C03641=1053.652,-40.489,430.295,170.687,30.205,155.689
C03642=1053.645,-40.738,430.307,170.685,30.204,155.689
C03643=1053.639,-40.988,430.320,170.683,30.202,155.688
C03644=1053.633,-41.237,430.333,170.681,30.201,155.688
C03645=1053.627,-41.487,430.346,170.680,30.199,155.688
C03646=1053.620,-41.736,430.359,170.678,30.197,155.688
C03647=1053.615,-41.986,430.372,170.676,30.195,155.688
C03648=1053.607,-42.236,430.385,170.674,30.194,155.687
C03649=1053.601,-42.485,430.397,170.672,30.192,155.687
C03650=1053.595,-42.735,430.410,170.670,30.191,155.687
C03651=1053.589,-42.985,430.423,170.669,30.189,155.687
C03652=1053.583,-43.234,430.436,170.667,30.188,155.687
C03653=1053.576,-43.483,430.448,170.665,30.185,155.687
C03654=1053.570,-43.733,430.461,170.663,30.184,155.686
C03655=1053.564,-43.983,430.474,170.661,30.182,155.686
C03656=1053.558,-44.233,430.487,170.660,30.181,155.686
C03657=1053.551,-44.482,430.499,170.658,30.179,155.686
C03658=1053.545,-44.731,430.512,170.656,30.178,155.686
C03659=1053.539,-44.981,430.524,170.654,30.176,155.686
C03660=1053.533,-45.230,430.538,170.652,30.174,155.685
C03661=1053.527,-45.480,430.550,170.650,30.172,155.685
C03662=1053.521,-45.730,430.562,170.649,30.171,155.685
C03663=1053.514,-45.979,430.575,170.647,30.169,155.685
C03664=1053.508,-46.229,430.588,170.645,30.168,155.685
C03665=1053.503,-46.479,430.601,170.643,30.166,155.685
C03666=1053.496,-46.728,430.613,170.641,30.164,155.684
C03667=1053.490,-46.978,430.626,170.639,30.163,155.684
C03668=1053.484,-47.228,430.638,170.638,30.161,155.684
C03669=1053.478,-47.478,430.651,170.636,30.160,155.684
C03670=1053.471,-47.727,430.664,170.634,30.158,155.684
C03671=1053.465,-47.976,430.676,170.632,30.157,155.684
C03672=1053.459,-48.226,430.689,170.630,30.154,155.683
C03673=1053.453,-48.476,430.702,170.628,30.153,155.683
C03674=1053.446,-48.725,430.714,170.627,30.151,155.683
C03675=1053.440,-48.975,430.726,170.625,30.150,155.683
C03676=1053.434,-49.225,430.739,170.623,30.148,155.683
C03677=1053.429,-49.474,430.751,170.621,30.147,155.683
C03678=1053.422,-49.723,430.764,170.619,30.145,155.682
C03679=1053.416,-49.973,430.776,170.617,30.143,155.682
C03680=1053.410,-50.223,430.789,170.616,30.142,155.682
C03681=1053.404,-50.504,430.803,170.613,30.140,155.682
C03682=1053.396,-50.783,430.817,170.611,30.139,155.682
C03683=1053.388,-51.064,430.831,170.609,30.137,155.682
C03684=1053.381,-51.344,430.845,170.607,30.135,155.681
C03685=1053.375,-51.594,430.857,170.605,30.134,155.681
C03686=1053.369,-51.844,430.869,170.604,30.132,155.681
C03687=1053.363,-52.093,430.881,170.601,30.130,155.681
C03688=1053.357,-52.343,430.893,170.599,30.129,155.681
C03689=1053.350,-52.592,430.905,170.597,30.127,155.681
C03690=1053.343,-52.841,430.918,170.595,30.126,155.681
C03691=1053.337,-53.091,430.931,170.593,30.125,155.680
C03692=1053.331,-53.341,430.943,170.592,30.123,155.680
C03693=1053.325,-53.590,430.955,170.590,30.122,155.680
C03694=1053.318,-53.840,430.967,170.588,30.120,155.680
C03695=1053.312,-54.090,430.980,170.586,30.119,155.680
C03696=1053.306,-54.339,430.992,170.584,30.118,155.680
C03697=1053.299,-54.589,431.003,170.582,30.116,155.680
C03698=1053.293,-54.839,431.016,170.581,30.114,155.679
C03699=1053.287,-55.088,431.028,170.579,30.113,155.679
C03700=1053.281,-55.338,431.041,170.577,30.112,155.679
C03701=1053.275,-55.587,431.052,170.575,30.110,155.679
C03702=1053.268,-55.837,431.064,170.573,30.109,155.679
C03703=1053.262,-56.087,431.077,170.571,30.107,155.679
C03704=1053.255,-56.336,431.089,170.570,30.106,155.679
C03705=1053.249,-56.586,431.101,170.568,30.105,155.679
C03706=1053.243,-56.836,431.113,170.566,30.103,155.678
C03707=1053.236,-57.085,431.125,170.564,30.101,155.678
C03708=1053.230,-57.335,431.138,170.561,30.100,155.678
C03709=1053.224,-57.584,431.149,170.559,30.099,155.678
C03710=1053.218,-57.834,431.161,170.557,30.097,155.678
C03711=1053.212,-58.084,431.174,170.556,30.096,155.678
C03712=1053.205,-58.334,431.185,170.554,30.094,155.678
C03713=1053.199,-58.583,431.197,170.552,30.093,155.678
C03714=1053.193,-58.833,431.210,170.550,30.091,155.677
C03715=1053.187,-59.082,431.221,170.548,30.090,155.677
C03716=1053.181,-59.332,431.234,170.546,30.088,155.677
C03717=1053.174,-59.581,431.246,170.545,30.087,155.677
C03718=1053.168,-59.831,431.258,170.543,30.086,155.677
C03719=1053.162,-60.081,431.270,170.541,30.084,155.677
C03720=1053.155,-60.331,431.281,170.539,30.083,155.677
C03721=1053.149,-60.580,431.293,170.537,30.082,155.677
C03722=1053.143,-60.830,431.306,170.535,30.080,155.676
C03723=1053.137,-61.079,431.317,170.534,30.079,155.676
C03724=1053.130,-61.329,431.329,170.532,30.078,155.676
C03725=1053.125,-61.578,431.342,170.530,30.076,155.676
C03726=1053.118,-61.828,431.353,170.527,30.074,155.676
C03727=1053.112,-62.078,431.365,170.525,30.073,155.676
C03728=1053.106,-62.328,431.377,170.523,30.072,155.676
C03729=1053.100,-62.577,431.389,170.521,30.070,155.676
C03730=1053.093,-62.827,431.400,170.520,30.069,155.675
C03731=1053.088,-63.077,431.413,170.518,30.068,155.675
C03732=1053.081,-63.326,431.425,170.516,30.066,155.675
C03733=1053.075,-63.575,431.436,170.514,30.064,155.675
C03734=1053.069,-63.826,431.448,170.512,30.063,155.675
C03735=1053.063,-64.075,431.460,170.510,30.062,155.675
C03736=1053.056,-64.325,431.472,170.509,30.060,155.675
C03737=1053.050,-64.574,431.484,170.507,30.059,155.675
C03738=1053.044,-64.824,431.496,170.505,30.058,155.675
C03739=1053.038,-65.074,431.507,170.503,30.056,155.674
C03740=1053.032,-65.323,431.519,170.500,30.055,155.674
C03741=1053.026,-65.573,431.531,170.498,30.053,155.674
C03742=1053.019,-65.823,431.543,170.496,30.052,155.674
C03743=1053.013,-66.072,431.554,170.495,30.051,155.674
C03744=1053.008,-66.322,431.566,170.493,30.049,155.674
C03745=1053.001,-66.570,431.578,170.491,30.048,155.674
C03746=1052.995,-66.819,431.590,170.489,30.047,155.674
C03747=1052.989,-67.068,431.601,170.487,30.045,155.674
C03748=1052.982,-67.317,431.613,170.485,30.044,155.673
C03749=1052.976,-67.565,431.625,170.484,30.043,155.673
C03750=1052.971,-67.813,431.636,170.482,30.042,155.673
C03751=1052.965,-68.062,431.648,170.480,30.040,155.673
C03752=1052.959,-68.311,431.660,170.478,30.038,155.673
C03753=1052.952,-68.560,431.671,170.476,30.038,155.673
C03754=1052.947,-68.810,431.683,170.474,30.036,155.673
C03755=1052.940,-69.060,431.695,170.471,30.035,155.673
C03756=1052.934,-69.310,431.706,170.470,30.033,155.673
C03757=1052.928,-69.559,431.718,170.468,30.032,155.672
C03758=1052.922,-69.809,431.730,170.466,30.031,155.672
C03759=1052.916,-70.058,431.741,170.464,30.029,155.672
C03760=1052.910,-70.308,431.753,170.462,30.028,155.672
C03761=1052.903,-70.558,431.764,170.460,30.027,155.672
C03762=1052.898,-70.807,431.777,170.459,30.026,155.672
C03763=1052.892,-71.057,431.788,170.457,30.024,155.672
C03764=1052.886,-71.306,431.799,170.455,30.023,155.672
C03765=1052.879,-71.556,431.811,170.453,30.021,155.672
C03766=1052.874,-71.806,431.823,170.451,30.020,155.671
C03767=1052.868,-72.056,431.834,170.448,30.019,155.671
C03768=1052.861,-72.305,431.846,170.447,30.017,155.671
C03769=1052.855,-72.555,431.857,170.445,30.016,155.671
C03770=1052.849,-72.805,431.868,170.443,30.015,155.671
C03771=1052.844,-73.054,431.880,170.441,30.014,155.671
C03772=1052.837,-73.304,431.892,170.439,30.012,155.671
C03773=1052.831,-73.553,431.903,170.437,30.011,155.671
C03774=1052.825,-73.803,431.914,170.435,30.009,155.671
C03775=1052.819,-74.052,431.926,170.434,30.008,155.671
C03776=1052.812,-74.302,431.937,170.432,30.007,155.671
C03777=1052.807,-74.552,431.948,170.430,30.006,155.671
C03778=1052.800,-74.802,431.960,170.427,30.005,155.670
C03779=1052.794,-75.052,431.971,170.425,30.003,155.670
C03780=1052.788,-75.301,431.982,170.423,30.002,155.670
C03781=1052.781,-75.551,431.994,170.421,30.001,155.670
C03782=1052.776,-75.800,432.005,170.420,30.000,155.670
C03783=1052.769,-76.050,432.016,170.418,29.999,155.670
C03784=1052.763,-76.299,432.028,170.416,29.998,155.670
C03785=1052.757,-76.550,432.039,170.414,29.996,155.670
C03786=1052.751,-76.799,432.050,170.412,29.995,155.670
C03787=1052.744,-77.049,432.062,170.409,29.994,155.670
C03788=1052.739,-77.298,432.073,170.407,29.992,155.670
C03789=1052.732,-77.582,432.085,170.406,29.991,155.670
C03790=1052.725,-77.866,432.098,170.403,29.990,155.670
C03791=1052.717,-78.149,432.112,170.401,29.989,155.669
C03792=1052.710,-78.433,432.124,170.399,29.988,155.669
C03793=1052.705,-78.683,432.135,170.397,29.986,155.669
C03794=1052.698,-78.933,432.146,170.394,29.985,155.669
C03795=1052.692,-79.182,432.158,170.392,29.984,155.669
C03796=1052.686,-79.432,432.169,170.391,29.982,155.669
C03797=1052.680,-79.682,432.180,170.389,29.981,155.669
C03798=1052.674,-79.931,432.191,170.387,29.981,155.669
C03799=1052.668,-80.181,432.202,170.385,29.980,155.669
C03800=1052.661,-80.430,432.213,170.383,29.979,155.669
C03801=1052.655,-80.680,432.224,170.381,29.978,155.669
C03802=1052.649,-80.930,432.236,170.378,29.976,155.669
C03803=1052.642,-81.180,432.246,170.377,29.975,155.669
C03804=1052.636,-81.430,432.257,170.375,29.974,155.669
C03805=1052.630,-81.679,432.268,170.373,29.973,155.669
C03806=1052.624,-81.929,432.279,170.371,29.972,155.669
C03807=1052.617,-82.179,432.290,170.369,29.971,155.669
C03808=1052.611,-82.427,432.301,170.367,29.970,155.668
C03809=1052.604,-82.711,432.314,170.364,29.969,155.668
C03810=1052.597,-82.995,432.326,170.363,29.967,155.668
C03811=1052.589,-83.279,432.338,170.360,29.966,155.668
C03812=1052.582,-83.563,432.351,170.358,29.965,155.668
C03813=1052.576,-83.813,432.362,170.356,29.964,155.668
C03814=1052.569,-84.063,432.373,170.354,29.963,155.668
C03815=1052.564,-84.312,432.384,170.352,29.962,155.668
C03816=1052.558,-84.562,432.394,170.349,29.961,155.668
C03817=1052.552,-84.812,432.406,170.347,29.960,155.668
C03818=1052.545,-85.061,432.416,170.346,29.959,155.668
C03819=1052.539,-85.311,432.427,170.344,29.958,155.668
C03820=1052.533,-85.561,432.438,170.342,29.957,155.668
C03821=1052.527,-85.810,432.448,170.340,29.956,155.668
C03822=1052.520,-86.060,432.460,170.338,29.955,155.668
C03823=1052.514,-86.309,432.470,170.335,29.954,155.668
C03824=1052.507,-86.559,432.481,170.333,29.953,155.668
C03825=1052.502,-86.809,432.492,170.331,29.952,155.668
C03826=1052.496,-87.058,432.503,170.330,29.951,155.668
C03827=1052.489,-87.308,432.514,170.328,29.950,155.668
C03828=1052.483,-87.558,432.524,170.326,29.949,155.668
C03829=1052.477,-87.808,432.535,170.324,29.948,155.668
C03830=1052.471,-88.058,432.545,170.321,29.947,155.668
C03831=1052.465,-88.307,432.556,170.319,29.946,155.668
C03832=1052.459,-88.557,432.567,170.317,29.945,155.668
C03833=1052.452,-88.807,432.578,170.315,29.944,155.668
C03834=1052.446,-89.056,432.588,170.314,29.943,155.667
C03835=1052.440,-89.306,432.600,170.312,29.942,155.667
C03836=1052.433,-89.555,432.610,170.309,29.941,155.667
C03837=1052.428,-89.805,432.621,170.307,29.940,155.667
C03838=1052.422,-90.056,432.631,170.305,29.939,155.667
C03839=1052.415,-90.305,432.642,170.303,29.938,155.667
C03840=1052.409,-90.554,432.653,170.301,29.937,155.667
C03841=1052.404,-90.804,432.663,170.300,29.936,155.667
C03842=1052.397,-91.054,432.674,170.298,29.935,155.667
C03843=1052.391,-91.303,432.685,170.295,29.934,155.667
C03844=1052.385,-91.553,432.695,170.293,29.933,155.667
C03845=1052.378,-91.803,432.706,170.291,29.932,155.667
C03846=1052.373,-92.053,432.717,170.289,29.932,155.667
C03847=1052.366,-92.302,432.727,170.287,29.931,155.667
C03848=1052.360,-92.551,432.738,170.285,29.930,155.667
C03849=1052.354,-92.802,432.748,170.283,29.929,155.667
C03850=1052.348,-93.051,432.759,170.281,29.928,155.667
C03851=1052.342,-93.301,432.770,170.279,29.927,155.667
C03852=1052.336,-93.550,432.780,170.277,29.926,155.667
C03853=1052.330,-93.801,432.790,170.275,29.925,155.667
C03854=1052.324,-94.050,432.801,170.273,29.924,155.667
C03855=1052.317,-94.299,432.811,170.271,29.923,155.667
C03856=1052.312,-94.550,432.822,170.268,29.922,155.667
C03857=1052.305,-94.799,432.832,170.267,29.921,155.667
C03858=1052.299,-95.049,432.843,170.265,29.920,155.667
C03859=1052.293,-95.298,432.854,170.263,29.919,155.667
C03860=1052.287,-95.548,432.864,170.261,29.918,155.667
C03861=1052.282,-95.798,432.874,170.259,29.918,155.667
C03862=1052.274,-96.048,432.885,170.257,29.917,155.667
C03863=1052.269,-96.298,432.895,170.254,29.916,155.667
C03864=1052.263,-96.547,432.906,170.252,29.915,155.667
C03865=1052.257,-96.796,432.916,170.250,29.914,155.667
C03866=1052.251,-97.047,432.927,170.249,29.913,155.667
C03867=1052.244,-97.296,432.937,170.247,29.912,155.667
C03868=1052.239,-97.547,432.947,170.245,29.911,155.667
C03869=1052.232,-97.796,432.958,170.242,29.910,155.667
C03870=1052.227,-98.045,432.969,170.240,29.910,155.667
C03871=1052.221,-98.295,432.978,170.238,29.909,155.667
C03872=1052.213,-98.545,432.989,170.236,29.908,155.667
C03873=1052.206,-98.831,433.000,170.233,29.907,155.667
C03874=1052.199,-99.117,433.012,170.232,29.906,155.667
C03875=1052.193,-99.403,433.024,170.229,29.905,155.667
C03876=1052.186,-99.689,433.036,170.227,29.904,155.667
C03877=1052.180,-99.939,433.045,170.225,29.904,155.667
C03878=1052.173,-100.189,433.056,170.223,29.903,155.667
C03879=1052.167,-100.438,433.067,170.220,29.902,155.667
C03880=1052.161,-100.688,433.076,170.218,29.901,155.667
C03881=1052.154,-100.937,433.087,170.216,29.901,155.667
C03882=1052.149,-101.187,433.097,170.214,29.900,155.667
C03883=1052.143,-101.437,433.106,170.213,29.899,155.667
C03884=1052.136,-101.687,433.117,170.211,29.899,155.667
C03885=1052.130,-101.937,433.127,170.208,29.898,155.667
C03886=1052.124,-102.186,433.138,170.206,29.897,155.667
C03887=1052.118,-102.436,433.147,170.204,29.896,155.667
C03888=1052.112,-102.686,433.158,170.202,29.895,155.667
C03889=1052.106,-102.935,433.168,170.200,29.895,155.667
C03890=1052.099,-103.185,433.178,170.197,29.894,155.667
C03891=1052.094,-103.435,433.188,170.195,29.893,155.667
C03892=1052.087,-103.685,433.198,170.194,29.892,155.667
C03893=1052.081,-103.934,433.208,170.192,29.892,155.667
C03894=1052.074,-104.184,433.218,170.190,29.891,155.667
C03895=1052.069,-104.434,433.229,170.188,29.891,155.667
C03896=1052.063,-104.683,433.238,170.185,29.890,155.667
C03897=1052.056,-104.933,433.248,170.183,29.889,155.667
C03898=1052.051,-105.183,433.259,170.181,29.888,155.667
C03899=1052.044,-105.433,433.268,170.179,29.888,155.667
C03900=1052.038,-105.682,433.278,170.177,29.887,155.667
C03901=1052.032,-105.931,433.288,170.174,29.886,155.667
C03902=1052.026,-106.182,433.298,170.173,29.885,155.667
C03903=1052.020,-106.431,433.308,170.171,29.885,155.667
C03904=1052.014,-106.681,433.318,170.169,29.884,155.667
C03905=1052.007,-106.931,433.328,170.167,29.884,155.667
C03906=1052.002,-107.181,433.338,170.165,29.883,155.667
C03907=1051.995,-107.431,433.348,170.162,29.882,155.667
C03908=1051.989,-107.680,433.358,170.160,29.882,155.668
C03909=1051.983,-107.930,433.368,170.158,29.881,155.667
C03910=1051.977,-108.180,433.377,170.156,29.880,155.668
C03911=1051.970,-108.430,433.387,170.154,29.879,155.668
C03912=1051.964,-108.679,433.397,170.152,29.879,155.668
C03913=1051.958,-108.929,433.407,170.150,29.879,155.668
C03914=1051.952,-109.179,433.417,170.148,29.878,155.668
C03915=1051.946,-109.428,433.426,170.146,29.877,155.668
C03916=1051.940,-109.678,433.436,170.144,29.877,155.668
C03917=1051.933,-109.927,433.446,170.141,29.876,155.668
C03918=1051.927,-110.177,433.456,170.139,29.875,155.668
C03919=1051.921,-110.427,433.465,170.137,29.875,155.668
C03920=1051.915,-110.677,433.475,170.135,29.875,155.668
C03921=1051.909,-110.927,433.484,170.133,29.874,155.668
C03922=1051.903,-111.176,433.495,170.131,29.873,155.668
C03923=1051.897,-111.426,433.505,170.129,29.873,155.668
C03924=1051.891,-111.676,433.514,170.127,29.872,155.668
C03925=1051.885,-111.926,433.524,170.125,29.871,155.668
C03926=1051.878,-112.175,433.534,170.123,29.871,155.668
C03927=1051.872,-112.425,433.543,170.120,29.870,155.668
C03928=1051.866,-112.675,433.553,170.118,29.869,155.668
C03929=1051.860,-112.925,433.562,170.116,29.869,155.668
C03930=1051.854,-113.174,433.572,170.114,29.869,155.668
C03931=1051.847,-113.424,433.582,170.112,29.868,155.669
C03932=1051.841,-113.673,433.592,170.109,29.867,155.669
C03933=1051.835,-113.923,433.601,170.108,29.867,155.669
C03934=1051.829,-114.173,433.611,170.106,29.866,155.669
C03935=1051.823,-114.423,433.621,170.104,29.866,155.669
C03936=1051.817,-114.673,433.631,170.102,29.866,155.669
C03937=1051.810,-114.957,433.641,170.099,29.865,155.669
C03938=1051.803,-115.242,433.651,170.097,29.864,155.669
C03939=1051.796,-115.526,433.663,170.094,29.864,155.669
C03940=1051.789,-115.811,433.673,170.092,29.863,155.669
C03941=1051.783,-116.061,433.683,170.089,29.863,155.669
C03942=1051.776,-116.311,433.693,170.087,29.862,155.669
C03943=1051.770,-116.561,433.702,170.085,29.862,155.669
C03944=1051.764,-116.811,433.712,170.083,29.862,155.669
C03945=1051.758,-117.060,433.721,170.082,29.861,155.669
C03946=1051.752,-117.310,433.730,170.079,29.860,155.670
C03947=1051.746,-117.559,433.740,170.077,29.860,155.670
C03948=1051.740,-117.809,433.750,170.075,29.859,155.670
C03949=1051.734,-118.060,433.758,170.073,29.859,155.670
C03950=1051.728,-118.309,433.768,170.071,29.859,155.670
C03951=1051.722,-118.559,433.778,170.068,29.858,155.670
C03952=1051.716,-118.809,433.787,170.066,29.858,155.670
C03953=1051.709,-119.058,433.796,170.064,29.857,155.670
C03954=1051.702,-119.308,433.806,170.062,29.857,155.670
C03955=1051.697,-119.557,433.815,170.060,29.857,155.670
C03956=1051.691,-119.807,433.824,170.057,29.856,155.670
C03957=1051.685,-120.057,433.834,170.056,29.856,155.670
C03958=1051.679,-120.307,433.843,170.054,29.855,155.670
C03959=1051.673,-120.557,433.852,170.052,29.855,155.671
C03960=1051.666,-120.807,433.862,170.049,29.855,155.671
C03961=1051.660,-121.057,433.872,170.047,29.854,155.671
C03962=1051.654,-121.306,433.880,170.045,29.854,155.671
C03963=1051.648,-121.555,433.890,170.043,29.853,155.671
C03964=1051.642,-121.806,433.899,170.041,29.853,155.671
C03965=1051.636,-122.056,433.908,170.038,29.853,155.671
C03966=1051.629,-122.305,433.918,170.036,29.852,155.671
C03967=1051.624,-122.554,433.927,170.034,29.852,155.671
C03968=1051.617,-122.804,433.936,170.032,29.851,155.671
C03969=1051.611,-123.054,433.945,170.030,29.851,155.671
C03970=1051.605,-123.304,433.954,170.028,29.851,155.671
C03971=1051.599,-123.554,433.964,170.026,29.850,155.672
C03972=1051.593,-123.803,433.973,170.024,29.850,155.672
C03973=1051.587,-124.053,433.982,170.022,29.850,155.672
C03974=1051.580,-124.303,433.991,170.020,29.850,155.672
C03975=1051.574,-124.553,434.000,170.017,29.849,155.672
C03976=1051.568,-124.803,434.009,170.015,29.849,155.672
C03977=1051.563,-125.052,434.018,170.013,29.848,155.672
C03978=1051.556,-125.302,434.027,170.011,29.848,155.672
C03979=1051.550,-125.552,434.036,170.008,29.848,155.672
C03980=1051.544,-125.802,434.046,170.006,29.848,155.672
C03981=1051.537,-126.051,434.055,170.004,29.847,155.673
C03982=1051.532,-126.301,434.063,170.002,29.847,155.673
C03983=1051.526,-126.551,434.073,170.000,29.847,155.673
C03984=1051.519,-126.801,434.082,169.998,29.847,155.673
C03985=1051.513,-127.051,434.091,169.996,29.846,155.673
C03986=1051.507,-127.300,434.100,169.994,29.846,155.673
C03987=1051.501,-127.550,434.109,169.992,29.846,155.673
C03988=1051.494,-127.800,434.118,169.989,29.845,155.673
C03989=1051.490,-128.049,434.128,169.987,29.845,155.673
C03990=1051.486,-128.299,434.138,169.985,29.844,155.673
C03991=1051.482,-128.550,434.148,169.983,29.842,155.673
C03992=1051.480,-128.799,434.159,169.981,29.840,155.673
C03993=1051.479,-129.050,434.172,169.981,29.837,155.672
C03994=1051.480,-129.301,434.185,169.979,29.834,155.672
C03995=1051.481,-129.551,434.198,169.977,29.830,155.672
C03996=1051.483,-129.801,434.213,169.977,29.826,155.671
C03997=1051.486,-130.052,434.227,169.975,29.822,155.670
C03998=1051.491,-130.302,434.243,169.975,29.817,155.669
C03999=1051.497,-130.553,434.259,169.974,29.811,155.668
C04000=1051.503,-130.803,434.275,169.974,29.805,155.667
C04001=1051.137,-130.826,434.054,169.927,29.973,155.700
C04002=1051.131,-130.577,434.037,169.928,29.980,155.701
C04003=1051.125,-130.326,434.021,169.928,29.985,155.702
C04004=1051.120,-130.076,434.006,169.929,29.990,155.703
C04005=1051.117,-129.824,433.990,169.930,29.995,155.703
C04006=1051.114,-129.574,433.977,169.931,29.999,155.704
C04007=1051.113,-129.324,433.962,169.933,30.003,155.704
C04008=1051.113,-129.074,433.951,169.934,30.006,155.705
C04009=1051.114,-128.823,433.938,169.935,30.008,155.705
C04010=1051.116,-128.573,433.927,169.937,30.010,155.705
C04011=1051.119,-128.323,433.916,169.939,30.012,155.706
C04012=1051.123,-128.073,433.905,169.941,30.013,155.706
C04013=1051.128,-127.823,433.897,169.943,30.014,155.706
C04014=1051.134,-127.573,433.887,169.945,30.015,155.706
C04015=1051.140,-127.324,433.878,169.947,30.014,155.705
C04016=1051.146,-127.074,433.870,169.949,30.015,155.705
C04017=1051.153,-126.824,433.860,169.951,30.015,155.705
C04018=1051.159,-126.575,433.851,169.954,30.016,155.705
C04019=1051.165,-126.324,433.842,169.956,30.015,155.705
C04020=1051.171,-126.075,433.833,169.958,30.016,155.705
C04021=1051.177,-125.826,433.823,169.960,30.016,155.705
C04022=1051.183,-125.575,433.815,169.962,30.016,155.705
C04023=1051.190,-125.326,433.806,169.965,30.017,155.705
C04024=1051.196,-125.076,433.796,169.967,30.017,155.704
C04025=1051.201,-124.826,433.788,169.969,30.017,155.704
C04026=1051.207,-124.576,433.778,169.971,30.017,155.704
C04027=1051.214,-124.327,433.769,169.974,30.018,155.704
C04028=1051.220,-124.076,433.760,169.976,30.018,155.704
C04029=1051.226,-123.827,433.751,169.977,30.019,155.704
C04030=1051.232,-123.577,433.741,169.979,30.019,155.704
C04031=1051.238,-123.328,433.732,169.981,30.019,155.704
C04032=1051.245,-123.078,433.724,169.984,30.019,155.704
C04033=1051.251,-122.828,433.714,169.986,30.020,155.704
C04034=1051.257,-122.579,433.705,169.988,30.020,155.704
C04035=1051.263,-122.329,433.695,169.990,30.020,155.703
C04036=1051.269,-122.078,433.686,169.993,30.021,155.703
C04037=1051.275,-121.829,433.677,169.995,30.021,155.703
C04038=1051.282,-121.579,433.668,169.997,30.021,155.703
C04039=1051.288,-121.329,433.658,169.999,30.022,155.703
C04040=1051.293,-121.080,433.649,170.001,30.022,155.703
C04041=1051.300,-120.831,433.640,170.004,30.023,155.703
C04042=1051.305,-120.580,433.631,170.006,30.023,155.703
C04043=1051.312,-120.330,433.621,170.007,30.023,155.703
C04044=1051.318,-120.080,433.612,170.009,30.024,155.703
C04045=1051.324,-119.831,433.602,170.012,30.024,155.703
C04046=1051.330,-119.582,433.593,170.014,30.025,155.703
C04047=1051.336,-119.332,433.584,170.016,30.025,155.703
C04048=1051.343,-119.082,433.574,170.018,30.025,155.702
C04049=1051.348,-118.832,433.565,170.020,30.026,155.702
C04050=1051.355,-118.582,433.556,170.023,30.026,155.702
C04051=1051.361,-118.332,433.546,170.025,30.027,155.702
C04052=1051.367,-118.082,433.537,170.027,30.027,155.702
C04053=1051.373,-117.833,433.527,170.029,30.027,155.702
C04054=1051.379,-117.583,433.518,170.031,30.028,155.702
C04055=1051.385,-117.334,433.508,170.034,30.028,155.702
C04056=1051.391,-117.084,433.499,170.035,30.029,155.702
C04057=1051.397,-116.834,433.489,170.037,30.030,155.702
C04058=1051.403,-116.584,433.480,170.039,30.030,155.702
C04059=1051.410,-116.335,433.471,170.042,30.030,155.702
C04060=1051.416,-116.085,433.461,170.044,30.031,155.702
C04061=1051.423,-115.835,433.452,170.046,30.031,155.701
C04062=1051.429,-115.550,433.440,170.048,30.031,155.701
C04063=1051.436,-115.265,433.430,170.051,30.032,155.701
C04064=1051.443,-114.980,433.419,170.054,30.033,155.701
C04065=1051.451,-114.696,433.408,170.056,30.034,155.701
C04066=1051.457,-114.446,433.398,170.058,30.034,155.701
C04067=1051.463,-114.197,433.389,170.059,30.034,155.701
C04068=1051.469,-113.947,433.379,170.062,30.035,155.701
C04069=1051.475,-113.697,433.370,170.064,30.035,155.701
C04070=1051.481,-113.448,433.360,170.066,30.036,155.701
C04071=1051.487,-113.197,433.350,170.068,30.036,155.701
C04072=1051.493,-112.948,433.341,170.070,30.037,155.701
C04073=1051.499,-112.698,433.331,170.073,30.037,155.701
C04074=1051.505,-112.448,433.321,170.075,30.038,155.701
C04075=1051.511,-112.198,433.312,170.077,30.039,155.701
C04076=1051.517,-111.948,433.302,170.079,30.039,155.701
C04077=1051.524,-111.699,433.292,170.081,30.039,155.701
C04078=1051.530,-111.449,433.282,170.083,30.041,155.701
C04079=1051.536,-111.200,433.273,170.085,30.041,155.700
C04080=1051.542,-110.950,433.263,170.087,30.041,155.700
C04081=1051.549,-110.700,433.254,170.089,30.042,155.700
C04082=1051.554,-110.450,433.244,170.091,30.043,155.700
C04083=1051.560,-110.200,433.234,170.094,30.043,155.700
C04084=1051.567,-109.951,433.224,170.096,30.043,155.700
C04085=1051.573,-109.701,433.214,170.098,30.044,155.700
C04086=1051.579,-109.451,433.205,170.100,30.045,155.700
C04087=1051.585,-109.202,433.195,170.102,30.045,155.700
C04088=1051.591,-108.952,433.185,170.105,30.046,155.700
C04089=1051.598,-108.703,433.175,170.107,30.047,155.700
C04090=1051.604,-108.453,433.166,170.108,30.047,155.700
C04091=1051.609,-108.203,433.155,170.110,30.048,155.700
C04092=1051.616,-107.953,433.146,170.112,30.048,155.700
C04093=1051.622,-107.704,433.136,170.115,30.049,155.700
C04094=1051.628,-107.454,433.126,170.117,30.050,155.700
C04095=1051.634,-107.204,433.116,170.119,30.050,155.700
C04096=1051.641,-106.954,433.107,170.121,30.051,155.700
C04097=1051.647,-106.704,433.096,170.123,30.051,155.700
C04098=1051.653,-106.454,433.086,170.126,30.052,155.700
C04099=1051.659,-106.205,433.077,170.128,30.053,155.700
C04100=1051.666,-105.955,433.066,170.129,30.053,155.700
C04101=1051.671,-105.705,433.056,170.131,30.054,155.700
C04102=1051.677,-105.455,433.047,170.133,30.055,155.700
C04103=1051.684,-105.206,433.036,170.136,30.056,155.700
C04104=1051.690,-104.956,433.027,170.138,30.056,155.700
C04105=1051.695,-104.706,433.017,170.140,30.057,155.700
C04106=1051.702,-104.457,433.006,170.142,30.057,155.699
C04107=1051.708,-104.207,432.997,170.144,30.058,155.700
C04108=1051.714,-103.958,432.986,170.147,30.059,155.699
C04109=1051.721,-103.707,432.976,170.149,30.060,155.699
C04110=1051.727,-103.458,432.966,170.150,30.060,155.699
C04111=1051.732,-103.208,432.955,170.152,30.061,155.699
C04112=1051.739,-102.958,432.946,170.154,30.062,155.699
C04113=1051.745,-102.709,432.936,170.156,30.063,155.699
C04114=1051.751,-102.459,432.926,170.159,30.063,155.699
C04115=1051.757,-102.209,432.916,170.161,30.064,155.699
C04116=1051.763,-101.960,432.906,170.163,30.064,155.699
C04117=1051.769,-101.710,432.896,170.165,30.065,155.699
C04118=1051.776,-101.460,432.885,170.167,30.066,155.699
C04119=1051.782,-101.210,432.875,170.170,30.067,155.699
C04120=1051.788,-100.961,432.865,170.171,30.068,155.699
C04121=1051.794,-100.711,432.855,170.173,30.068,155.699
C04122=1051.800,-100.462,432.844,170.175,30.069,155.699
C04123=1051.806,-100.212,432.835,170.177,30.070,155.699
C04124=1051.813,-99.962,432.824,170.179,30.071,155.699
C04125=1051.819,-99.712,432.814,170.182,30.072,155.699
C04126=1051.826,-99.426,432.802,170.184,30.072,155.699
C04127=1051.833,-99.140,432.791,170.187,30.073,155.699
C04128=1051.840,-98.854,432.779,170.189,30.074,155.699
C04129=1051.848,-98.567,432.767,170.191,30.075,155.699
C04130=1051.853,-98.318,432.756,170.193,30.076,155.699
C04131=1051.860,-98.069,432.746,170.195,30.077,155.699
C04132=1051.865,-97.819,432.736,170.197,30.078,155.699
C04133=1051.872,-97.569,432.726,170.199,30.078,155.699
C04134=1051.879,-97.319,432.716,170.202,30.079,155.699
C04135=1051.884,-97.069,432.705,170.204,30.080,155.699
C04136=1051.890,-96.820,432.694,170.206,30.080,155.699
C04137=1051.896,-96.570,432.685,170.208,30.081,155.699
C04138=1051.902,-96.321,432.674,170.209,30.082,155.699
C04139=1051.909,-96.071,432.663,170.211,30.083,155.699
C04140=1051.914,-95.821,432.653,170.213,30.084,155.699
C04141=1051.920,-95.571,432.642,170.216,30.085,155.699
C04142=1051.927,-95.322,432.632,170.218,30.086,155.699
C04143=1051.932,-95.072,432.622,170.220,30.087,155.699
C04144=1051.939,-94.822,432.611,170.222,30.088,155.699
C04145=1051.945,-94.573,432.600,170.224,30.089,155.699
C04146=1051.951,-94.323,432.590,170.225,30.090,155.699
C04147=1051.957,-94.073,432.580,170.228,30.091,155.699
C04148=1051.963,-93.824,432.569,170.230,30.091,155.699
C04149=1051.970,-93.574,432.558,170.232,30.092,155.699
C04150=1051.975,-93.324,432.548,170.234,30.093,155.699
C04151=1051.981,-93.074,432.537,170.236,30.094,155.699
C04152=1051.987,-92.825,432.527,170.238,30.095,155.699
C04153=1051.994,-92.575,432.515,170.241,30.096,155.699
C04154=1052.000,-92.325,432.506,170.243,30.097,155.700
C04155=1052.006,-92.076,432.495,170.244,30.098,155.700
C04156=1052.012,-91.825,432.484,170.246,30.099,155.700
C04157=1052.018,-91.576,432.473,170.248,30.099,155.700
C04158=1052.024,-91.327,432.463,170.250,30.100,155.700
C04159=1052.030,-91.077,432.452,170.252,30.101,155.700
C04160=1052.037,-90.827,432.442,170.255,30.103,155.700
C04161=1052.042,-90.577,432.431,170.257,30.103,155.700
C04162=1052.049,-90.328,432.421,170.259,30.104,155.700
C04163=1052.055,-90.078,432.409,170.260,30.105,155.700
C04164=1052.061,-89.828,432.399,170.262,30.106,155.700
C04165=1052.067,-89.579,432.389,170.264,30.107,155.700
C04166=1052.073,-89.328,432.378,170.267,30.108,155.700
C04167=1052.079,-89.079,432.367,170.269,30.109,155.700
C04168=1052.086,-88.830,432.357,170.271,30.110,155.700
C04169=1052.092,-88.580,432.345,170.273,30.111,155.700
C04170=1052.098,-88.330,432.334,170.275,30.112,155.700
C04171=1052.104,-88.081,432.324,170.276,30.113,155.700
C04172=1052.111,-87.831,432.313,170.278,30.114,155.700
C04173=1052.116,-87.581,432.302,170.281,30.115,155.700
C04174=1052.123,-87.332,432.292,170.283,30.116,155.700
C04175=1052.129,-87.082,432.280,170.285,30.117,155.700
C04176=1052.135,-86.832,432.270,170.287,30.118,155.700
C04177=1052.142,-86.582,432.260,170.289,30.119,155.700
C04178=1052.147,-86.332,432.249,170.291,30.120,155.700
C04179=1052.153,-86.083,432.238,170.293,30.121,155.700
C04180=1052.160,-85.833,432.227,170.295,30.122,155.700
C04181=1052.166,-85.584,432.216,170.297,30.123,155.700
C04182=1052.172,-85.333,432.205,170.299,30.124,155.700
C04183=1052.179,-85.084,432.195,170.301,30.125,155.700
C04184=1052.184,-84.835,432.184,170.303,30.126,155.701
C04185=1052.191,-84.584,432.173,170.305,30.127,155.701
C04186=1052.197,-84.335,432.162,170.308,30.128,155.701
C04187=1052.204,-84.086,432.151,170.310,30.129,155.701
C04188=1052.210,-83.836,432.140,170.311,30.130,155.701
C04189=1052.216,-83.586,432.128,170.313,30.131,155.701
C04190=1052.223,-83.303,432.117,170.315,30.132,155.701
C04191=1052.230,-83.019,432.104,170.318,30.133,155.701
C04192=1052.237,-82.735,432.091,170.320,30.134,155.701
C04193=1052.244,-82.451,432.079,170.323,30.136,155.701
C04194=1052.251,-82.202,432.068,170.325,30.137,155.701
C04195=1052.257,-81.952,432.057,170.326,30.138,155.701
C04196=1052.263,-81.702,432.046,170.328,30.139,155.701
C04197=1052.269,-81.452,432.035,170.330,30.140,155.701
C04198=1052.276,-81.203,432.025,170.332,30.141,155.701
C04199=1052.282,-80.953,432.014,170.335,30.142,155.701
C04200=1052.288,-80.703,432.003,170.337,30.143,155.701
C04201=1052.294,-80.454,431.991,170.339,30.144,155.701
C04202=1052.301,-80.204,431.980,170.341,30.145,155.701
C04203=1052.307,-79.954,431.969,170.342,30.146,155.701
C04204=1052.313,-79.705,431.958,170.344,30.147,155.701
C04205=1052.319,-79.454,431.947,170.346,30.148,155.702
C04206=1052.325,-79.205,431.936,170.348,30.149,155.702
C04207=1052.332,-78.955,431.924,170.351,30.151,155.702
C04208=1052.337,-78.706,431.913,170.353,30.152,155.702
C04209=1052.344,-78.456,431.902,170.355,30.153,155.702
C04210=1052.349,-78.206,431.891,170.357,30.154,155.702
C04211=1052.356,-77.957,431.879,170.358,30.155,155.702
C04212=1052.363,-77.707,431.869,170.360,30.157,155.702
C04213=1052.369,-77.457,431.858,170.362,30.158,155.702
C04214=1052.375,-77.208,431.847,170.364,30.159,155.702
C04215=1052.381,-76.958,431.835,170.366,30.160,155.702
C04216=1052.387,-76.709,431.824,170.369,30.161,155.702
C04217=1052.393,-76.459,431.813,170.371,30.162,155.702
C04218=1052.399,-76.210,431.801,170.372,30.164,155.702
C04219=1052.406,-75.959,431.790,170.374,30.165,155.702
C04220=1052.412,-75.709,431.779,170.376,30.166,155.703
C04221=1052.418,-75.460,431.767,170.378,30.167,155.703
C04222=1052.425,-75.210,431.756,170.380,30.168,155.703
C04223=1052.430,-74.961,431.745,170.382,30.169,155.703
C04224=1052.437,-74.711,431.733,170.384,30.170,155.703
C04225=1052.443,-74.462,431.722,170.386,30.172,155.703
C04226=1052.449,-74.211,431.711,170.388,30.173,155.703
C04227=1052.456,-73.962,431.699,170.390,30.174,155.703
C04228=1052.461,-73.712,431.688,170.392,30.175,155.703
C04229=1052.467,-73.463,431.676,170.394,30.177,155.703
C04230=1052.473,-73.213,431.665,170.396,30.178,155.703
C04231=1052.480,-72.963,431.653,170.398,30.180,155.704
C04232=1052.485,-72.714,431.642,170.400,30.180,155.704
C04233=1052.492,-72.464,431.631,170.401,30.182,155.704
C04234=1052.497,-72.215,431.618,170.403,30.183,155.704
C04235=1052.503,-71.964,431.607,170.406,30.185,155.704
C04236=1052.509,-71.716,431.596,170.408,30.186,155.704
C04237=1052.516,-71.465,431.584,170.410,30.187,155.704
C04238=1052.522,-71.215,431.572,170.412,30.188,155.704
C04239=1052.527,-70.966,431.561,170.413,30.190,155.704
C04240=1052.534,-70.716,431.549,170.415,30.191,155.704
C04241=1052.540,-70.467,431.538,170.417,30.192,155.705
C04242=1052.546,-70.217,431.525,170.419,30.193,155.705
C04243=1052.551,-69.968,431.515,170.421,30.195,155.705
C04244=1052.558,-69.718,431.503,170.423,30.196,155.705
C04245=1052.565,-69.468,431.491,170.425,30.197,155.705
C04246=1052.570,-69.219,431.479,170.426,30.199,155.705
C04247=1052.576,-68.969,431.467,170.429,30.200,155.705
C04248=1052.583,-68.719,431.456,170.431,30.202,155.705
C04249=1052.589,-68.470,431.444,170.433,30.203,155.705
C04250=1052.594,-68.219,431.433,170.435,30.204,155.705
C04251=1052.600,-67.971,431.421,170.437,30.206,155.706
C04252=1052.607,-67.721,431.409,170.439,30.207,155.706
C04253=1052.613,-67.471,431.397,170.440,30.208,155.706
C04254=1052.620,-67.189,431.384,170.442,30.210,155.706
C04255=1052.627,-66.907,431.371,170.445,30.211,155.706
C04256=1052.633,-66.626,431.357,170.447,30.213,155.706
C04257=1052.641,-66.344,431.344,170.449,30.214,155.706
C04258=1052.646,-66.095,431.333,170.452,30.216,155.706
C04259=1052.653,-65.845,431.321,170.453,30.217,155.706
C04260=1052.659,-65.595,431.309,170.455,30.218,155.707
C04261=1052.664,-65.346,431.297,170.457,30.219,155.707
C04262=1052.671,-65.096,431.285,170.459,30.221,155.707
C04263=1052.678,-64.846,431.273,170.461,30.223,155.707
C04264=1052.683,-64.597,431.263,170.463,30.224,155.707
C04265=1052.689,-64.347,431.250,170.465,30.225,155.707
C04266=1052.696,-64.098,431.238,170.466,30.227,155.707
C04267=1052.703,-63.848,431.226,170.468,30.228,155.707
C04268=1052.708,-63.598,431.215,170.470,30.229,155.708
C04269=1052.714,-63.349,431.203,170.472,30.231,155.708
C04270=1052.721,-63.099,431.191,170.474,30.232,155.708
C04271=1052.726,-62.850,431.179,170.476,30.233,155.708
C04272=1052.733,-62.600,431.167,170.479,30.235,155.708
C04273=1052.739,-62.350,431.155,170.480,30.236,155.708
C04274=1052.745,-62.100,431.143,170.482,30.238,155.708
C04275=1052.752,-61.851,431.131,170.484,30.239,155.708
C04276=1052.758,-61.602,431.119,170.486,30.240,155.708
C04277=1052.763,-61.351,431.107,170.488,30.242,155.709
C04278=1052.770,-61.102,431.095,170.490,30.243,155.709
C04279=1052.777,-60.852,431.084,170.492,30.244,155.709
C04280=1052.782,-60.603,431.071,170.493,30.246,155.709
C04281=1052.789,-60.353,431.059,170.495,30.247,155.709
C04282=1052.795,-60.104,431.047,170.497,30.248,155.709
C04283=1052.801,-59.853,431.036,170.499,30.250,155.709
C04284=1052.808,-59.604,431.024,170.501,30.251,155.709
C04285=1052.814,-59.355,431.012,170.503,30.253,155.710
C04286=1052.820,-59.105,430.999,170.504,30.254,155.710
C04287=1052.826,-58.855,430.987,170.506,30.256,155.710
C04288=1052.833,-58.606,430.976,170.509,30.257,155.710
C04289=1052.839,-58.356,430.963,170.511,30.259,155.710
C04290=1052.845,-58.106,430.951,170.513,30.260,155.710
C04291=1052.851,-57.857,430.939,170.515,30.261,155.710
C04292=1052.857,-57.607,430.928,170.517,30.263,155.710
C04293=1052.864,-57.357,430.916,170.518,30.264,155.710
C04294=1052.870,-57.108,430.903,170.520,30.265,155.711
C04295=1052.876,-56.858,430.891,170.522,30.267,155.711
C04296=1052.883,-56.608,430.879,170.524,30.269,155.711
C04297=1052.889,-56.358,430.867,170.526,30.270,155.711
C04298=1052.895,-56.110,430.855,170.528,30.271,155.711
C04299=1052.902,-55.861,430.842,170.530,30.273,155.711
C04300=1052.907,-55.612,430.830,170.531,30.274,155.711
C04301=1052.914,-55.362,430.818,170.533,30.276,155.712
C04302=1052.920,-55.112,430.806,170.535,30.277,155.712
C04303=1052.927,-54.864,430.794,170.537,30.278,155.712
C04304=1052.933,-54.614,430.781,170.539,30.280,155.712
C04305=1052.939,-54.365,430.770,170.541,30.281,155.712
C04306=1052.945,-54.116,430.758,170.542,30.282,155.712
C04307=1052.951,-53.866,430.745,170.544,30.284,155.712
C04308=1052.958,-53.616,430.733,170.547,30.286,155.712
C04309=1052.964,-53.366,430.721,170.549,30.287,155.713
C04310=1052.971,-53.117,430.709,170.551,30.289,155.713
C04311=1052.977,-52.867,430.697,170.553,30.290,155.713
C04312=1052.983,-52.618,430.684,170.555,30.291,155.713
C04313=1052.990,-52.369,430.672,170.556,30.293,155.713
C04314=1052.996,-52.119,430.659,170.558,30.295,155.713
C04315=1053.003,-51.869,430.647,170.560,30.296,155.713
C04316=1053.008,-51.619,430.635,170.562,30.297,155.714
C04317=1053.015,-51.370,430.623,170.564,30.299,155.714
C04318=1053.022,-51.089,430.609,170.566,30.300,155.714
C04319=1053.030,-50.808,430.595,170.567,30.302,155.714
C04320=1053.036,-50.526,430.581,170.570,30.303,155.714
C04321=1053.044,-50.245,430.567,170.572,30.306,155.714
C04322=1053.050,-49.995,430.554,170.574,30.307,155.715
C04323=1053.056,-49.746,430.542,170.576,30.309,155.715
C04324=1053.063,-49.496,430.529,170.578,30.310,155.715
C04325=1053.068,-49.247,430.517,170.579,30.312,155.715
C04326=1053.074,-48.997,430.504,170.581,30.313,155.715
C04327=1053.080,-48.748,430.492,170.583,30.315,155.715
C04328=1053.087,-48.498,430.479,170.585,30.317,155.716
C04329=1053.093,-48.249,430.467,170.587,30.318,155.716
C04330=1053.098,-47.999,430.454,170.589,30.320,155.716
C04331=1053.105,-47.749,430.442,170.591,30.321,155.716
C04332=1053.111,-47.500,430.429,170.592,30.323,155.716
C04333=1053.117,-47.250,430.416,170.594,30.324,155.716
C04334=1053.123,-47.000,430.404,170.596,30.326,155.716
C04335=1053.130,-46.751,430.391,170.598,30.328,155.717
C04336=1053.136,-46.501,430.378,170.600,30.329,155.717
C04337=1053.142,-46.251,430.366,170.602,30.331,155.717
C04338=1053.148,-46.002,430.353,170.603,30.333,155.717
C04339=1053.154,-45.752,430.340,170.605,30.334,155.717
C04340=1053.161,-45.503,430.328,170.607,30.336,155.718
C04341=1053.167,-45.253,430.315,170.609,30.337,155.718
C04342=1053.173,-45.003,430.302,170.611,30.339,155.718
C04343=1053.179,-44.754,430.290,170.613,30.341,155.718
C04344=1053.186,-44.505,430.277,170.614,30.342,155.718
C04345=1053.192,-44.255,430.265,170.616,30.344,155.718
C04346=1053.197,-44.005,430.252,170.618,30.345,155.718
C04347=1053.204,-43.756,430.239,170.620,30.347,155.719
C04348=1053.210,-43.506,430.226,170.622,30.349,155.719
C04349=1053.217,-43.257,430.213,170.624,30.351,155.719
C04350=1053.222,-43.007,430.201,170.625,30.352,155.719
C04351=1053.229,-42.758,430.188,170.627,30.354,155.719
C04352=1053.235,-42.508,430.175,170.629,30.355,155.720
C04353=1053.240,-42.258,430.163,170.631,30.357,155.720
C04354=1053.248,-42.008,430.150,170.633,30.358,155.720
C04355=1053.254,-41.758,430.137,170.635,30.360,155.720
C04356=1053.260,-41.509,430.124,170.636,30.362,155.720
C04357=1053.266,-41.259,430.111,170.638,30.364,155.720
C04358=1053.272,-41.010,430.098,170.640,30.365,155.721
C04359=1053.278,-40.760,430.085,170.642,30.367,155.721
C04360=1053.285,-40.511,430.073,170.644,30.368,155.721
C04361=1053.291,-40.261,430.060,170.646,30.370,155.721
C04362=1053.297,-40.012,430.047,170.648,30.371,155.721
C04363=1053.303,-39.762,430.034,170.649,30.374,155.722
C04364=1053.310,-39.512,430.021,170.651,30.375,155.722
C04365=1053.317,-39.262,430.009,170.653,30.377,155.722
C04366=1053.323,-39.013,429.995,170.655,30.378,155.722
C04367=1053.329,-38.764,429.982,170.657,30.380,155.722
C04368=1053.335,-38.514,429.970,170.659,30.381,155.722
C04369=1053.341,-38.265,429.956,170.660,30.384,155.723
C04370=1053.347,-38.015,429.944,170.662,30.385,155.723
C04371=1053.353,-37.766,429.930,170.664,30.387,155.723
C04372=1053.360,-37.516,429.917,170.666,30.389,155.723
C04373=1053.366,-37.266,429.904,170.668,30.390,155.723
C04374=1053.372,-37.017,429.891,170.670,30.392,155.724
C04375=1053.378,-36.767,429.878,170.671,30.394,155.724
C04376=1053.384,-36.517,429.865,170.673,30.396,155.724
C04377=1053.390,-36.268,429.851,170.675,30.397,155.724
C04378=1053.396,-36.018,429.839,170.677,30.399,155.724
C04379=1053.402,-35.769,429.826,170.679,30.401,155.725
C04380=1053.409,-35.519,429.812,170.681,30.403,155.725
C04381=1053.415,-35.269,429.799,170.681,30.404,155.725
C04382=1053.422,-34.989,429.784,170.684,30.406,155.725
C04383=1053.429,-34.710,429.769,170.686,30.408,155.725
C04384=1053.436,-34.430,429.755,170.688,30.410,155.726
C04385=1053.443,-34.150,429.740,170.690,30.412,155.726
C04386=1053.449,-33.900,429.727,170.691,30.414,155.726
C04387=1053.455,-33.651,429.714,170.693,30.415,155.726
C04388=1053.461,-33.401,429.701,170.695,30.417,155.726
C04389=1053.468,-33.151,429.687,170.697,30.419,155.727
C04390=1053.474,-32.902,429.675,170.699,30.421,155.727
C04391=1053.480,-32.652,429.661,170.701,30.423,155.727
C04392=1053.485,-32.403,429.647,170.702,30.424,155.727
C04393=1053.492,-32.153,429.634,170.704,30.426,155.728
C04394=1053.498,-31.904,429.621,170.706,30.428,155.728
C04395=1053.504,-31.654,429.608,170.708,30.429,155.728
C04396=1053.511,-31.404,429.595,170.710,30.432,155.728
C04397=1053.517,-31.155,429.581,170.712,30.433,155.728
C04398=1053.524,-30.905,429.568,170.713,30.435,155.728
C04399=1053.530,-30.656,429.555,170.715,30.437,155.729
C04400=1053.536,-30.407,429.541,170.717,30.438,155.729
C04401=1053.542,-30.157,429.529,170.718,30.440,155.729
C04402=1053.548,-29.906,429.514,170.720,30.442,155.729
C04403=1053.554,-29.657,429.501,170.722,30.444,155.729
C04404=1053.560,-29.408,429.488,170.723,30.446,155.730
C04405=1053.567,-29.159,429.475,170.725,30.447,155.730
C04406=1053.573,-28.909,429.461,170.727,30.449,155.730
C04407=1053.580,-28.659,429.448,170.729,30.451,155.730
C04408=1053.586,-28.410,429.435,170.731,30.453,155.731
C04409=1053.592,-28.160,429.422,170.733,30.454,155.731
C04410=1053.598,-27.910,429.408,170.734,30.456,155.731
C04411=1053.604,-27.661,429.394,170.736,30.458,155.731
C04412=1053.611,-27.411,429.381,170.738,30.460,155.731
C04413=1053.617,-27.162,429.368,170.740,30.462,155.732
C04414=1053.623,-26.912,429.354,170.742,30.463,155.732
C04415=1053.630,-26.663,429.341,170.744,30.465,155.732
C04416=1053.636,-26.413,429.327,170.744,30.467,155.732
C04417=1053.642,-26.163,429.314,170.746,30.469,155.732
C04418=1053.648,-25.914,429.300,170.748,30.471,155.733
C04419=1053.654,-25.664,429.286,170.750,30.472,155.733
C04420=1053.660,-25.415,429.273,170.752,30.475,155.733
C04421=1053.666,-25.165,429.259,170.754,30.476,155.733
C04422=1053.672,-24.916,429.246,170.755,30.478,155.734
C04423=1053.679,-24.666,429.232,170.757,30.480,155.734
C04424=1053.684,-24.416,429.218,170.759,30.482,155.734
C04425=1053.691,-24.167,429.205,170.761,30.484,155.734
C04426=1053.697,-23.917,429.191,170.763,30.486,155.735
C04427=1053.703,-23.668,429.177,170.765,30.487,155.735
C04428=1053.709,-23.419,429.163,170.765,30.489,155.735
C04429=1053.716,-23.169,429.150,170.767,30.491,155.735
C04430=1053.722,-22.919,429.136,170.769,30.493,155.735
C04431=1053.728,-22.670,429.123,170.771,30.495,155.736
C04432=1053.734,-22.420,429.108,170.773,30.497,155.736
C04433=1053.740,-22.170,429.095,170.775,30.499,155.736
C04434=1053.746,-21.921,429.082,170.776,30.500,155.736
C04435=1053.752,-21.671,429.068,170.778,30.503,155.737
C04436=1053.759,-21.422,429.054,170.780,30.505,155.737
C04437=1053.764,-21.173,429.040,170.782,30.506,155.737
C04438=1053.771,-20.923,429.026,170.784,30.508,155.737
C04439=1053.777,-20.673,429.013,170.785,30.510,155.737
C04440=1053.784,-20.423,428.999,170.786,30.512,155.738
C04441=1053.790,-20.175,428.985,170.788,30.513,155.738
C04442=1053.796,-19.925,428.971,170.790,30.516,155.738
C04443=1053.802,-19.675,428.957,170.792,30.518,155.738
C04444=1053.809,-19.426,428.944,170.794,30.519,155.739
C04445=1053.815,-19.175,428.930,170.796,30.521,155.739
C04446=1053.822,-18.895,428.915,170.797,30.524,155.739
C04447=1053.829,-18.615,428.898,170.799,30.526,155.739
C04448=1053.836,-18.334,428.883,170.801,30.527,155.740
C04449=1053.842,-18.053,428.867,170.803,30.529,155.740
C04450=1053.849,-17.803,428.854,170.805,30.532,155.740
C04451=1053.856,-17.555,428.840,170.806,30.534,155.740
C04452=1053.862,-17.305,428.825,170.808,30.535,155.741
C04453=1053.868,-17.055,428.812,170.810,30.537,155.741
C04454=1053.874,-16.805,428.798,170.812,30.539,155.741
C04455=1053.880,-16.556,428.784,170.814,30.541,155.741
C04456=1053.886,-16.306,428.770,170.816,30.543,155.742
C04457=1053.893,-16.057,428.756,170.816,30.545,155.742
C04458=1053.899,-15.808,428.742,170.818,30.547,155.742
C04459=1053.905,-15.558,428.728,170.820,30.548,155.742
C04460=1053.912,-15.309,428.715,170.822,30.551,155.743
C04461=1053.918,-15.059,428.700,170.824,30.553,155.743
C04462=1053.923,-14.809,428.686,170.826,30.554,155.743
C04463=1053.930,-14.559,428.672,170.827,30.556,155.743
C04464=1053.936,-14.310,428.658,170.829,30.559,155.744
C04465=1053.943,-14.060,428.644,170.831,30.561,155.744
C04466=1053.949,-13.812,428.630,170.832,30.562,155.744
C04467=1053.955,-13.561,428.615,170.834,30.564,155.744
C04468=1053.961,-13.312,428.602,170.836,30.566,155.745
C04469=1053.967,-13.062,428.587,170.837,30.569,155.745
C04470=1053.973,-12.813,428.573,170.839,30.570,155.745
C04471=1053.979,-12.564,428.559,170.841,30.572,155.745
C04472=1053.985,-12.314,428.545,170.843,30.574,155.746
C04473=1053.991,-12.065,428.531,170.844,30.576,155.746
C04474=1053.998,-11.815,428.517,170.846,30.578,155.746
C04475=1054.004,-11.566,428.502,170.847,30.580,155.746
C04476=1054.010,-11.316,428.488,170.849,30.582,155.747
C04477=1054.016,-11.067,428.474,170.851,30.584,155.747
C04478=1054.022,-10.817,428.460,170.853,30.586,155.747
C04479=1054.028,-10.568,428.445,170.855,30.588,155.747
C04480=1054.035,-10.318,428.432,170.855,30.590,155.748
C04481=1054.041,-10.069,428.417,170.857,30.592,155.748
C04482=1054.047,-9.819,428.403,170.859,30.594,155.748
C04483=1054.053,-9.569,428.388,170.861,30.596,155.748
C04484=1054.059,-9.320,428.375,170.863,30.598,155.749
C04485=1054.066,-9.070,428.360,170.865,30.600,155.749
C04486=1054.071,-8.820,428.346,170.866,30.602,155.749
C04487=1054.078,-8.571,428.332,170.867,30.604,155.749
C04488=1054.084,-8.322,428.317,170.869,30.606,155.750
C04489=1054.090,-8.072,428.303,170.871,30.608,155.750
C04490=1054.097,-7.823,428.289,170.873,30.610,155.750
C04491=1054.103,-7.573,428.275,170.875,30.612,155.750
C04492=1054.109,-7.323,428.260,170.876,30.614,155.751
C04493=1054.115,-7.074,428.245,170.878,30.616,155.751
C04494=1054.122,-6.824,428.231,170.879,30.618,155.751
C04495=1054.128,-6.575,428.217,170.881,30.619,155.751
C04496=1054.134,-6.326,428.202,170.883,30.622,155.752
C04497=1054.141,-6.076,428.188,170.885,30.624,155.752
C04498=1054.147,-5.827,428.174,170.886,30.626,155.752
C04499=1054.153,-5.577,428.159,170.888,30.628,155.753
C04500=1054.158,-5.328,428.145,170.890,30.630,155.753
C04501=1054.166,-5.078,428.130,170.891,30.632,155.753
C04502=1054.172,-4.829,428.115,170.893,30.634,155.753
C04503=1054.177,-4.579,428.102,170.895,30.636,155.754
C04504=1054.184,-4.329,428.087,170.896,30.638,155.754
C04505=1054.191,-4.080,428.072,170.898,30.639,155.754
C04506=1054.196,-3.830,428.058,170.900,30.642,155.754
C04507=1054.203,-3.581,428.044,170.901,30.644,155.755
C04508=1054.209,-3.331,428.029,170.903,30.646,155.755
C04509=1054.215,-3.082,428.014,170.905,30.648,155.755
C04510=1054.221,-2.799,427.998,170.906,30.650,155.755
C04511=1054.228,-2.517,427.981,170.908,30.652,155.756
C04512=1054.236,-2.235,427.965,170.910,30.655,155.756
C04513=1054.243,-1.953,427.948,170.912,30.657,155.756
C04514=1054.249,-1.704,427.934,170.914,30.659,155.757
C04515=1054.255,-1.454,427.919,170.915,30.661,155.757
C04516=1054.261,-1.204,427.905,170.917,30.663,155.757
C04517=1054.267,-0.955,427.890,170.919,30.666,155.757
C04518=1054.274,-0.705,427.875,170.920,30.668,155.758
C04519=1054.279,-0.456,427.860,170.922,30.670,155.758
C04520=1054.285,-0.206,427.845,170.924,30.672,155.758
C04521=1054.291,0.043,427.830,170.925,30.674,155.759
C04522=1054.297,0.292,427.815,170.927,30.676,155.759
C04523=1054.304,0.542,427.800,170.928,30.678,155.759
C04524=1054.310,0.792,427.786,170.930,30.680,155.760
C04525=1054.315,1.041,427.771,170.932,30.682,155.760
C04526=1054.322,1.291,427.757,170.934,30.685,155.760
C04527=1054.328,1.541,427.742,170.935,30.687,155.760
C04528=1054.334,1.790,427.727,170.937,30.689,155.761
C04529=1054.340,2.039,427.712,170.938,30.691,155.761
C04530=1054.347,2.289,427.697,170.940,30.693,155.761
C04531=1054.352,2.538,427.683,170.942,30.695,155.761
C04532=1054.359,2.788,427.668,170.943,30.697,155.762
C04533=1054.365,3.037,427.653,170.945,30.699,155.762
C04534=1054.371,3.286,427.638,170.946,30.701,155.762
C04535=1054.377,3.536,427.623,170.948,30.703,155.763
C04536=1054.384,3.785,427.608,170.950,30.706,155.763
C04537=1054.390,4.035,427.593,170.952,30.708,155.763
C04538=1054.395,4.284,427.578,170.953,30.710,155.763
C04539=1054.402,4.534,427.563,170.954,30.712,155.764
C04540=1054.408,4.784,427.548,170.956,30.714,155.764
C04541=1054.414,5.033,427.534,170.958,30.716,155.764
C04542=1054.420,5.282,427.519,170.960,30.718,155.765
C04543=1054.427,5.532,427.504,170.962,30.720,155.765
C04544=1054.433,5.782,427.489,170.962,30.722,155.765
C04545=1054.439,6.031,427.474,170.964,30.724,155.765
C04546=1054.445,6.280,427.459,170.966,30.726,155.766
C04547=1054.451,6.530,427.444,170.968,30.728,155.766
C04548=1054.458,6.780,427.429,170.970,30.730,155.766
C04549=1054.463,7.029,427.414,170.971,30.732,155.767
C04550=1054.469,7.278,427.399,170.972,30.734,155.767
C04551=1054.476,7.528,427.384,170.974,30.737,155.767
C04552=1054.482,7.777,427.369,170.976,30.739,155.767
C04553=1054.489,8.027,427.354,170.978,30.741,155.768
C04554=1054.495,8.276,427.339,170.979,30.743,155.768
C04555=1054.501,8.525,427.324,170.981,30.745,155.768
C04556=1054.507,8.775,427.309,170.982,30.747,155.769
C04557=1054.514,9.025,427.294,170.984,30.749,155.769
C04558=1054.519,9.275,427.279,170.986,30.751,155.769
C04559=1054.526,9.524,427.263,170.987,30.753,155.769
C04560=1054.532,9.773,427.248,170.989,30.755,155.770
C04561=1054.538,10.022,427.233,170.991,30.758,155.770
C04562=1054.545,10.272,427.219,170.992,30.760,155.770
C04563=1054.551,10.522,427.204,170.994,30.762,155.771
C04564=1054.558,10.771,427.188,170.995,30.764,155.771
C04565=1054.564,11.020,427.173,170.997,30.766,155.771
C04566=1054.569,11.270,427.158,170.999,30.768,155.771
C04567=1054.575,11.519,427.143,171.001,30.770,155.772
C04568=1054.582,11.769,427.128,171.001,30.772,155.772
C04569=1054.589,12.018,427.112,171.003,30.774,155.772
C04570=1054.595,12.268,427.097,171.005,30.776,155.773
C04571=1054.601,12.517,427.082,171.007,30.779,155.773
C04572=1054.608,12.767,427.067,171.009,30.781,155.773
C04573=1054.614,13.016,427.051,171.010,30.783,155.773
C04574=1054.621,13.300,427.035,171.011,30.785,155.774
C04575=1054.628,13.584,427.017,171.013,30.787,155.774
C04576=1054.635,13.869,427.000,171.016,30.790,155.775
C04577=1054.642,14.153,426.982,171.018,30.792,155.775
C04578=1054.648,14.402,426.967,171.019,30.794,155.775
C04579=1054.655,14.652,426.952,171.021,30.797,155.775
C04580=1054.661,14.901,426.936,171.022,30.799,155.776
C04581=1054.667,15.151,426.921,171.024,30.801,155.776
C04582=1054.673,15.401,426.906,171.025,30.803,155.776
C04583=1054.679,15.650,426.890,171.027,30.806,155.777
C04584=1054.686,15.900,426.875,171.029,30.808,155.777
C04585=1054.692,16.148,426.860,171.031,30.810,155.777
C04586=1054.697,16.398,426.844,171.031,30.812,155.778
C04587=1054.704,16.648,426.829,171.033,30.814,155.778
C04588=1054.710,16.897,426.813,171.035,30.816,155.778
C04589=1054.716,17.147,426.798,171.037,30.818,155.778
C04590=1054.723,17.396,426.782,171.039,30.821,155.779
C04591=1054.728,17.646,426.767,171.040,30.823,155.779
C04592=1054.735,17.895,426.751,171.041,30.825,155.779
C04593=1054.741,18.145,426.736,171.043,30.827,155.780
C04594=1054.747,18.394,426.721,171.045,30.829,155.780
C04595=1054.754,18.643,426.705,171.046,30.831,155.780
C04596=1054.759,18.893,426.690,171.048,30.833,155.781
C04597=1054.766,19.142,426.674,171.050,30.835,155.781
C04598=1054.771,19.392,426.659,171.051,30.838,155.781
C04599=1054.778,19.641,426.643,171.052,30.840,155.782
C04600=1054.784,19.890,426.628,171.054,30.842,155.782
C04601=1054.790,20.140,426.612,171.056,30.844,155.782
C04602=1054.797,20.389,426.597,171.058,30.847,155.782
C04603=1054.803,20.639,426.580,171.059,30.848,155.783
C04604=1054.809,20.888,426.565,171.060,30.851,155.783
C04605=1054.815,21.138,426.549,171.062,30.853,155.783
C04606=1054.821,21.387,426.533,171.064,30.855,155.784
C04607=1054.827,21.637,426.518,171.065,30.857,155.784
C04608=1054.833,21.886,426.502,171.067,30.860,155.784
C04609=1054.840,22.136,426.487,171.069,30.862,155.785
C04610=1054.846,22.385,426.471,171.070,30.864,155.785
C04611=1054.852,22.634,426.455,171.071,30.866,155.785
C04612=1054.858,22.884,426.439,171.073,30.868,155.786
C04613=1054.865,23.133,426.424,171.075,30.871,155.786
C04614=1054.870,23.383,426.408,171.077,30.873,155.786
C04615=1054.877,23.632,426.393,171.078,30.875,155.787
C04616=1054.883,23.881,426.376,171.079,30.877,155.787
C04617=1054.889,24.131,426.361,171.081,30.880,155.787
C04618=1054.895,24.380,426.345,171.083,30.882,155.787
C04619=1054.901,24.630,426.329,171.084,30.884,155.788
C04620=1054.907,24.879,426.314,171.086,30.886,155.788
C04621=1054.913,25.129,426.298,171.088,30.888,155.788
C04622=1054.920,25.378,426.282,171.089,30.891,155.789
C04623=1054.926,25.628,426.266,171.090,30.893,155.789
C04624=1054.932,25.877,426.251,171.092,30.895,155.789
C04625=1054.938,26.126,426.234,171.094,30.897,155.790
C04626=1054.944,26.375,426.218,171.096,30.900,155.790
C04627=1054.951,26.625,426.203,171.097,30.901,155.790
C04628=1054.957,26.874,426.187,171.098,30.904,155.791
C04629=1054.963,27.124,426.171,171.100,30.906,155.791
C04630=1054.969,27.373,426.155,171.102,30.908,155.791
C04631=1054.975,27.623,426.140,171.103,30.910,155.792
C04632=1054.982,27.872,426.124,171.105,30.913,155.792
C04633=1054.988,28.121,426.108,171.107,30.915,155.792
C04634=1054.994,28.371,426.091,171.107,30.917,155.793
C04635=1055.000,28.620,426.076,171.109,30.919,155.793
C04636=1055.006,28.870,426.060,171.111,30.921,155.793
C04637=1055.012,29.120,426.044,171.113,30.924,155.793
C04638=1055.019,29.405,426.025,171.115,30.926,155.794
C04639=1055.026,29.691,426.007,171.117,30.929,155.794
C04640=1055.034,29.976,425.989,171.118,30.932,155.795
C04641=1055.041,30.261,425.970,171.120,30.934,155.795
C04642=1055.046,30.511,425.955,171.121,30.936,155.795
C04643=1055.052,30.760,425.939,171.123,30.938,155.796
C04644=1055.058,31.009,425.922,171.125,30.941,155.796
C04645=1055.064,31.259,425.906,171.126,30.943,155.796
C04646=1055.071,31.508,425.890,171.127,30.945,155.797
C04647=1055.077,31.758,425.874,171.129,30.947,155.797
C04648=1055.083,32.007,425.857,171.131,30.950,155.797
C04649=1055.089,32.257,425.841,171.132,30.952,155.798
C04650=1055.096,32.506,425.826,171.134,30.954,155.798
C04651=1055.102,32.755,425.809,171.136,30.957,155.798
C04652=1055.108,33.005,425.794,171.137,30.959,155.799
C04653=1055.114,33.254,425.778,171.138,30.961,155.799
C04654=1055.120,33.504,425.761,171.140,30.963,155.799
C04655=1055.126,33.753,425.746,171.142,30.966,155.800
C04656=1055.133,34.003,425.729,171.143,30.968,155.800
C04657=1055.139,34.252,425.713,171.145,30.970,155.800
C04658=1055.145,34.501,425.696,171.146,30.973,155.801
C04659=1055.151,34.751,425.680,171.148,30.975,155.801
C04660=1055.157,35.000,425.664,171.149,30.977,155.801
C04661=1055.163,35.249,425.648,171.151,30.979,155.801
C04662=1055.169,35.499,425.632,171.153,30.982,155.802
C04663=1055.176,35.749,425.615,171.155,30.984,155.802
C04664=1055.182,35.998,425.599,171.156,30.986,155.802
C04665=1055.188,36.247,425.583,171.157,30.988,155.803
C04666=1055.194,36.497,425.567,171.159,30.990,155.803
C04667=1055.201,36.745,425.550,171.160,30.992,155.803
C04668=1055.207,36.995,425.534,171.162,30.994,155.804
C04669=1055.213,37.244,425.517,171.164,30.997,155.804
C04670=1055.219,37.494,425.501,171.166,30.999,155.804
C04671=1055.225,37.743,425.485,171.166,31.001,155.805
C04672=1055.231,37.993,425.469,171.168,31.004,155.805
C04673=1055.237,38.242,425.452,171.170,31.006,155.805
C04674=1055.243,38.492,425.436,171.171,31.008,155.806
C04675=1055.249,38.741,425.419,171.173,31.011,155.806
C04676=1055.256,38.990,425.403,171.175,31.013,155.806
C04677=1055.262,39.239,425.386,171.176,31.016,155.807
C04678=1055.268,39.489,425.370,171.177,31.018,155.807
C04679=1055.274,39.739,425.353,171.179,31.020,155.807
C04680=1055.280,39.988,425.337,171.181,31.022,155.808
C04681=1055.286,40.237,425.321,171.182,31.024,155.808
C04682=1055.292,40.486,425.304,171.184,31.026,155.808
C04683=1055.298,40.735,425.288,171.186,31.029,155.809
C04684=1055.304,40.985,425.271,171.187,31.031,155.809
C04685=1055.311,41.235,425.255,171.188,31.034,155.810
C04686=1055.317,41.484,425.239,171.190,31.036,155.810
C04687=1055.323,41.733,425.222,171.192,31.038,155.810
C04688=1055.329,41.982,425.205,171.193,31.041,155.811
C04689=1055.335,42.232,425.189,171.195,31.043,155.811
C04690=1055.341,42.482,425.172,171.196,31.045,155.811
C04691=1055.348,42.730,425.155,171.198,31.047,155.812
C04692=1055.353,42.980,425.139,171.199,31.049,155.812
C04693=1055.359,43.230,425.122,171.201,31.052,155.812
C04694=1055.365,43.480,425.106,171.203,31.054,155.813
C04695=1055.372,43.728,425.089,171.204,31.056,155.813
C04696=1055.378,43.978,425.072,171.205,31.059,155.813
C04697=1055.384,44.228,425.056,171.207,31.061,155.814
C04698=1055.390,44.477,425.038,171.208,31.064,155.814
C04699=1055.396,44.726,425.022,171.210,31.066,155.814
C04700=1055.402,44.975,425.006,171.212,31.068,155.815
C04701=1055.407,45.224,424.988,171.214,31.070,155.815
C04702=1055.415,45.510,424.969,171.215,31.073,155.815
C04703=1055.421,45.796,424.950,171.216,31.076,155.816
C04704=1055.428,46.081,424.931,171.218,31.078,155.816
C04705=1055.435,46.367,424.911,171.220,31.081,155.817
C04706=1055.441,46.616,424.895,171.222,31.084,155.817
C04707=1055.447,46.865,424.878,171.224,31.086,155.817
C04708=1055.454,47.115,424.861,171.224,31.089,155.818
C04709=1055.459,47.365,424.844,171.226,31.091,155.818
C04710=1055.465,47.613,424.827,171.228,31.093,155.818
C04711=1055.471,47.863,424.811,171.229,31.095,155.819
C04712=1055.477,48.112,424.793,171.231,31.098,155.819
C04713=1055.483,48.362,424.777,171.233,31.100,155.819
C04714=1055.489,48.610,424.760,171.235,31.103,155.820
C04715=1055.495,48.861,424.743,171.235,31.105,155.820
C04716=1055.501,49.109,424.726,171.237,31.107,155.821
C04717=1055.507,49.359,424.709,171.239,31.110,155.821
C04718=1055.514,49.608,424.693,171.240,31.112,155.821
C04719=1055.520,49.858,424.675,171.242,31.114,155.822
C04720=1055.526,50.107,424.658,171.244,31.117,155.822
C04721=1055.532,50.356,424.642,171.244,31.119,155.822
C04722=1055.538,50.606,424.624,171.246,31.122,155.823
C04723=1055.544,50.855,424.608,171.248,31.124,155.823
C04724=1055.550,51.104,424.591,171.249,31.126,155.823
C04725=1055.556,51.354,424.574,171.251,31.128,155.824
C04726=1055.562,51.603,424.557,171.253,31.130,155.824
C04727=1055.568,51.852,424.540,171.255,31.133,155.824
C04728=1055.574,52.102,424.523,171.255,31.135,155.825
C04729=1055.580,52.351,424.506,171.257,31.138,155.825
C04730=1055.586,52.600,424.489,171.259,31.140,155.825
C04731=1055.593,52.850,424.471,171.260,31.142,155.826
C04732=1055.598,53.099,424.455,171.262,31.144,155.826
C04733=1055.605,53.349,424.437,171.264,31.147,155.826
C04734=1055.611,53.598,424.420,171.265,31.149,155.827
C04735=1055.617,53.847,424.404,171.266,31.152,155.827
C04736=1055.623,54.097,424.386,171.268,31.154,155.828
C04737=1055.629,54.345,424.369,171.270,31.157,155.828
C04738=1055.636,54.596,424.352,171.271,31.159,155.828
C04739=1055.641,54.845,424.335,171.273,31.161,155.829
C04740=1055.647,55.094,424.319,171.275,31.163,155.829
C04741=1055.654,55.343,424.301,171.275,31.165,155.829
C04742=1055.660,55.592,424.284,171.277,31.168,155.830
C04743=1055.666,55.842,424.266,171.279,31.170,155.830
C04744=1055.672,56.091,424.250,171.280,31.173,155.830
C04745=1055.678,56.340,424.233,171.282,31.175,155.831
C04746=1055.685,56.590,424.215,171.284,31.177,155.831
C04747=1055.690,56.839,424.198,171.285,31.179,155.831
C04748=1055.697,57.089,424.181,171.286,31.181,155.832
C04749=1055.703,57.337,424.164,171.288,31.184,155.832
C04750=1055.709,57.587,424.146,171.290,31.186,155.832
C04751=1055.715,57.837,424.130,171.291,31.189,155.833
C04752=1055.721,58.086,424.112,171.293,31.191,155.833
C04753=1055.728,58.335,424.095,171.295,31.194,155.833
C04754=1055.734,58.584,424.078,171.296,31.196,155.834
C04755=1055.740,58.834,424.061,171.297,31.198,155.834
C04756=1055.746,59.084,424.043,171.299,31.200,155.834
C04757=1055.752,59.333,424.026,171.300,31.202,155.835
C04758=1055.759,59.582,424.009,171.302,31.205,155.835
C04759=1055.765,59.831,423.992,171.304,31.207,155.836
C04760=1055.771,60.081,423.974,171.306,31.210,155.836
C04761=1055.777,60.330,423.957,171.307,31.212,155.836
C04762=1055.783,60.580,423.939,171.308,31.214,155.837
C04763=1055.790,60.828,423.922,171.310,31.217,155.837
C04764=1055.796,61.078,423.905,171.311,31.218,155.837
C04765=1055.802,61.327,423.888,171.313,31.221,155.838
C04766=1055.809,61.613,423.868,171.315,31.224,155.838
C04767=1055.816,61.898,423.849,171.317,31.226,155.838
C04768=1055.823,62.183,423.828,171.318,31.229,155.839
C04769=1055.830,62.468,423.809,171.320,31.231,155.839
C04770=1055.836,62.718,423.791,171.322,31.234,155.840
C04771=1055.843,62.966,423.774,171.323,31.236,155.840
C04772=1055.849,63.216,423.756,171.325,31.238,155.840
C04773=1055.856,63.465,423.739,171.327,31.241,155.841
C04774=1055.861,63.714,423.721,171.328,31.243,155.841
C04775=1055.868,63.964,423.704,171.329,31.245,155.841
C04776=1055.874,64.213,423.687,171.331,31.247,155.842
C04777=1055.880,64.462,423.669,171.333,31.250,155.842
C04778=1055.886,64.711,423.651,171.334,31.252,155.842
C04779=1055.893,64.961,423.634,171.336,31.255,155.843
C04780=1055.898,65.210,423.616,171.338,31.257,155.843
C04781=1055.904,65.460,423.599,171.339,31.259,155.843
C04782=1055.911,65.709,423.581,171.340,31.262,155.844
C04783=1055.917,65.958,423.564,171.342,31.264,155.844
C04784=1055.923,66.208,423.546,171.343,31.266,155.844
C04785=1055.929,66.457,423.529,171.345,31.269,155.845
C04786=1055.935,66.706,423.511,171.347,31.271,155.845
C04787=1055.941,66.955,423.493,171.348,31.273,155.846
C04788=1055.947,67.205,423.475,171.350,31.276,155.846
C04789=1055.953,67.454,423.458,171.351,31.278,155.846
C04790=1055.959,67.704,423.440,171.352,31.280,155.847
C04791=1055.965,67.953,423.422,171.354,31.283,155.847
C04792=1055.972,68.202,423.405,171.356,31.286,155.847
C04793=1055.978,68.452,423.388,171.358,31.288,155.848
C04794=1055.984,68.700,423.369,171.359,31.290,155.848
C04795=1055.990,68.950,423.351,171.361,31.292,155.848
C04796=1055.996,69.199,423.334,171.362,31.295,155.849
C04797=1056.002,69.448,423.316,171.363,31.297,155.849
C04798=1056.008,69.698,423.299,171.365,31.300,155.850
C04799=1056.014,69.947,423.281,171.367,31.302,155.850
C04800=1056.020,70.197,423.263,171.368,31.304,155.850
C04801=1056.027,70.445,423.245,171.370,31.306,155.851
C04802=1056.033,70.695,423.227,171.372,31.309,155.851
C04803=1056.039,70.945,423.209,171.372,31.312,155.851
C04804=1056.044,71.194,423.192,171.374,31.314,155.852
C04805=1056.050,71.443,423.174,171.376,31.316,155.852
C04806=1056.056,71.692,423.156,171.378,31.318,155.852
C04807=1056.062,71.941,423.138,171.379,31.321,155.853
C04808=1056.069,72.191,423.120,171.381,31.323,155.853
C04809=1056.075,72.440,423.103,171.383,31.326,155.854
C04810=1056.081,72.689,423.084,171.383,31.328,155.854
C04811=1056.087,72.939,423.066,171.385,31.330,155.854
C04812=1056.093,73.188,423.049,171.387,31.333,155.855
C04813=1056.099,73.438,423.031,171.388,31.335,155.855
C04814=1056.105,73.686,423.012,171.390,31.338,155.855
C04815=1056.111,73.936,422.995,171.392,31.340,155.856
C04816=1056.117,74.185,422.977,171.393,31.342,155.856
C04817=1056.123,74.434,422.958,171.394,31.345,155.857
C04818=1056.129,74.684,422.940,171.396,31.347,155.857
C04819=1056.136,74.933,422.923,171.398,31.350,155.857
C04820=1056.142,75.181,422.905,171.399,31.352,155.858
C04821=1056.148,75.431,422.887,171.401,31.354,155.858
C04822=1056.154,75.681,422.869,171.403,31.357,155.858
C04823=1056.160,75.929,422.851,171.404,31.359,155.859
C04824=1056.166,76.179,422.833,171.405,31.362,155.859
C04825=1056.172,76.429,422.815,171.407,31.364,155.859
C04826=1056.178,76.677,422.796,171.408,31.366,155.860
C04827=1056.184,76.927,422.779,171.410,31.368,155.860
C04828=1056.190,77.176,422.760,171.412,31.371,155.861
C04829=1056.196,77.426,422.742,171.413,31.373,155.861
C04830=1056.203,77.710,422.722,171.415,31.376,155.861
C04831=1056.210,77.996,422.701,171.417,31.379,155.862
C04832=1056.218,78.281,422.680,171.418,31.382,155.862
C04833=1056.224,78.566,422.659,171.420,31.384,155.863
C04834=1056.230,78.815,422.641,171.422,31.387,155.863
C04835=1056.236,79.065,422.623,171.424,31.389,155.863
C04836=1056.242,79.313,422.605,171.425,31.391,155.864
C04837=1056.248,79.563,422.587,171.427,31.394,155.864
C04838=1056.254,79.812,422.568,171.429,31.396,155.864
C04839=1056.260,80.061,422.550,171.429,31.399,155.865
C04840=1056.266,80.311,422.531,171.431,31.401,155.865
C04841=1056.272,80.560,422.513,171.433,31.404,155.866
C04842=1056.278,80.809,422.495,171.434,31.406,155.866
C04843=1056.284,81.059,422.477,171.436,31.408,155.866
C04844=1056.290,81.308,422.458,171.438,31.411,155.867
C04845=1056.297,81.557,422.440,171.440,31.413,155.867
C04846=1056.301,81.806,422.422,171.440,31.415,155.867
C04847=1056.308,82.055,422.403,171.442,31.418,155.868
C04848=1056.314,82.305,422.385,171.444,31.421,155.868
C04849=1056.320,82.554,422.366,171.445,31.423,155.869
C04850=1056.326,82.803,422.349,171.447,31.425,155.869
C04851=1056.332,83.053,422.330,171.449,31.428,155.869
C04852=1056.338,83.302,422.311,171.450,31.430,155.870
C04853=1056.344,83.551,422.293,171.451,31.433,155.870
C04854=1056.350,83.800,422.275,171.453,31.435,155.871
C04855=1056.356,84.049,422.256,171.454,31.437,155.871
C04856=1056.362,84.299,422.237,171.456,31.440,155.871
C04857=1056.368,84.548,422.219,171.458,31.442,155.872
C04858=1056.374,84.797,422.201,171.460,31.445,155.872
C04859=1056.380,85.046,422.183,171.461,31.447,155.872
C04860=1056.387,85.295,422.164,171.463,31.449,155.873
C04861=1056.392,85.545,422.145,171.464,31.452,155.873
C04862=1056.398,85.795,422.127,171.465,31.454,155.874
C04863=1056.404,86.043,422.109,171.467,31.457,155.874
C04864=1056.411,86.292,422.090,171.469,31.459,155.874
C04865=1056.417,86.542,422.072,171.471,31.461,155.875
C04866=1056.422,86.791,422.053,171.472,31.464,155.875
C04867=1056.429,87.040,422.034,171.474,31.466,155.875
C04868=1056.435,87.290,422.016,171.476,31.469,155.876
C04869=1056.441,87.539,421.998,171.476,31.471,155.876
C04870=1056.447,87.788,421.979,171.478,31.473,155.876
C04871=1056.453,88.037,421.960,171.480,31.476,155.877
C04872=1056.459,88.286,421.941,171.481,31.478,155.877
C04873=1056.465,88.536,421.923,171.483,31.480,155.878
C04874=1056.472,88.785,421.905,171.485,31.483,155.878
C04875=1056.478,89.035,421.885,171.487,31.485,155.878
C04876=1056.483,89.283,421.867,171.487,31.488,155.879
C04877=1056.489,89.533,421.849,171.489,31.490,155.879
C04878=1056.496,89.782,421.831,171.491,31.492,155.879
C04879=1056.502,90.031,421.811,171.492,31.495,155.880
C04880=1056.508,90.280,421.793,171.494,31.497,155.880
C04881=1056.514,90.530,421.774,171.496,31.500,155.881
C04882=1056.520,90.779,421.755,171.498,31.502,155.881
C04883=1056.527,91.028,421.736,171.499,31.504,155.881
C04884=1056.531,91.277,421.718,171.500,31.507,155.882
C04885=1056.538,91.527,421.699,171.502,31.510,155.882
C04886=1056.544,91.776,421.681,171.503,31.512,155.883
C04887=1056.550,92.025,421.661,171.505,31.514,155.883
C04888=1056.556,92.274,421.643,171.507,31.517,155.883
C04889=1056.562,92.524,421.624,171.509,31.520,155.884
C04890=1056.568,92.773,421.605,171.510,31.521,155.884
C04891=1056.574,93.022,421.586,171.512,31.524,155.884
C04892=1056.580,93.271,421.567,171.513,31.527,155.885
C04893=1056.586,93.520,421.548,171.514,31.529,155.885
C04894=1056.592,93.806,421.527,171.516,31.532,155.886
C04895=1056.600,94.090,421.505,171.518,31.535,155.886
C04896=1056.607,94.375,421.484,171.520,31.537,155.887
C04897=1056.613,94.660,421.462,171.522,31.540,155.887
C04898=1056.619,94.910,421.442,171.524,31.543,155.887
C04899=1056.626,95.159,421.424,171.525,31.545,155.888
C04900=1056.631,95.408,421.404,171.526,31.547,155.888
C04901=1056.637,95.657,421.386,171.528,31.550,155.888
C04902=1056.643,95.906,421.367,171.530,31.553,155.889
C04903=1056.649,96.155,421.348,171.532,31.555,155.889
C04904=1056.655,96.405,421.329,171.533,31.557,155.890
C04905=1056.661,96.654,421.310,171.535,31.560,155.890
C04906=1056.667,96.903,421.291,171.537,31.562,155.890
C04907=1056.673,97.152,421.272,171.537,31.564,155.891
C04908=1056.679,97.402,421.253,171.539,31.567,155.891
C04909=1056.685,97.651,421.235,171.541,31.569,155.891
C04910=1056.691,97.900,421.215,171.543,31.572,155.892
C04911=1056.698,98.149,421.196,171.544,31.574,155.892
C04912=1056.704,98.398,421.177,171.546,31.576,155.893
C04913=1056.710,98.647,421.158,171.548,31.579,155.893
C04914=1056.716,98.897,421.139,171.549,31.582,155.893
C04915=1056.722,99.146,421.120,171.551,31.584,155.894
C04916=1056.728,99.395,421.101,171.552,31.586,155.894
C04917=1056.734,99.645,421.082,171.554,31.589,155.895
C04918=1056.740,99.893,421.062,171.555,31.591,155.895
C04919=1056.746,100.143,421.043,171.557,31.594,155.895
C04920=1056.752,100.392,421.024,171.559,31.596,155.896
C04921=1056.758,100.641,421.005,171.561,31.598,155.896
C04922=1056.764,100.891,420.987,171.562,31.601,155.897
C04923=1056.770,101.140,420.967,171.564,31.603,155.897
C04924=1056.776,101.389,420.947,171.565,31.606,155.897
C04925=1056.782,101.638,420.928,171.567,31.608,155.898
C04926=1056.788,101.887,420.909,171.568,31.611,155.898
C04927=1056.794,102.137,420.890,171.570,31.613,155.898
C04928=1056.800,102.386,420.870,171.572,31.616,155.899
C04929=1056.806,102.635,420.851,171.573,31.618,155.899
C04930=1056.811,102.884,420.832,171.575,31.621,155.900
C04931=1056.818,103.133,420.812,171.577,31.623,155.900
C04932=1056.824,103.382,420.793,171.578,31.626,155.900
C04933=1056.829,103.632,420.774,171.579,31.628,155.901
C04934=1056.835,103.881,420.754,171.581,31.630,155.901
C04935=1056.842,104.130,420.735,171.583,31.633,155.902
C04936=1056.848,104.379,420.716,171.585,31.636,155.902
C04937=1056.854,104.628,420.696,171.586,31.638,155.902
C04938=1056.859,104.877,420.677,171.588,31.640,155.903
C04939=1056.865,105.127,420.658,171.590,31.643,155.903
C04940=1056.872,105.375,420.638,171.590,31.645,155.904
C04941=1056.877,105.625,420.619,171.592,31.648,155.904
C04942=1056.883,105.874,420.600,171.594,31.650,155.904
C04943=1056.889,106.123,420.580,171.596,31.653,155.905
C04944=1056.895,106.372,420.561,171.597,31.655,155.905
C04945=1056.901,106.621,420.541,171.599,31.657,155.905
C04946=1056.908,106.871,420.522,171.601,31.660,155.906
C04947=1056.913,107.121,420.502,171.603,31.663,155.906
C04948=1056.919,107.369,420.482,171.604,31.665,155.907
C04949=1056.925,107.619,420.463,171.605,31.667,155.907
C04950=1056.931,107.868,420.443,171.607,31.670,155.907
C04951=1056.938,108.117,420.425,171.609,31.673,155.908
C04952=1056.944,108.365,420.405,171.610,31.675,155.908
C04953=1056.949,108.615,420.385,171.612,31.677,155.909
C04954=1056.955,108.864,420.365,171.614,31.680,155.909
C04955=1056.961,109.113,420.346,171.616,31.682,155.909
C04956=1056.967,109.363,420.326,171.617,31.684,155.910
C04957=1056.974,109.612,420.307,171.618,31.687,155.910
C04958=1056.980,109.897,420.285,171.620,31.690,155.911
C04959=1056.987,110.181,420.262,171.622,31.692,155.911
C04960=1056.994,110.466,420.240,171.624,31.695,155.911
C04961=1057.001,110.752,420.218,171.626,31.698,155.912
C04962=1057.007,111.001,420.198,171.628,31.700,155.912
C04963=1057.013,111.250,420.178,171.630,31.703,155.913
C04964=1057.019,111.499,420.158,171.632,31.706,155.913
C04965=1057.025,111.748,420.138,171.633,31.708,155.914
C04966=1057.031,111.997,420.119,171.634,31.710,155.914
C04967=1057.037,112.246,420.099,171.636,31.713,155.914
C04968=1057.043,112.496,420.079,171.638,31.715,155.915
C04969=1057.049,112.745,420.060,171.639,31.718,155.915
C04970=1057.055,112.994,420.040,171.641,31.720,155.915
C04971=1057.061,113.243,420.020,171.643,31.723,155.916
C04972=1057.067,113.492,420.001,171.645,31.725,155.916
C04973=1057.073,113.741,419.981,171.646,31.728,155.917
C04974=1057.079,113.991,419.961,171.648,31.730,155.917
C04975=1057.085,114.240,419.941,171.649,31.733,155.917
C04976=1057.091,114.489,419.921,171.651,31.735,155.918
C04977=1057.097,114.738,419.902,171.652,31.738,155.918
C04978=1057.102,114.987,419.881,171.654,31.740,155.919
C04979=1057.108,115.236,419.861,171.656,31.743,155.919
C04980=1057.114,115.485,419.841,171.658,31.746,155.920
C04981=1057.120,115.735,419.822,171.659,31.748,155.920
C04982=1057.125,115.984,419.801,171.661,31.750,155.920
C04983=1057.131,116.233,419.781,171.662,31.753,155.921
C04984=1057.137,116.482,419.761,171.664,31.755,155.921
C04985=1057.143,116.731,419.741,171.665,31.758,155.922
C04986=1057.148,116.981,419.721,171.667,31.761,155.922
C04987=1057.155,117.230,419.701,171.669,31.763,155.922
C04988=1057.161,117.479,419.681,171.671,31.766,155.923
C04989=1057.167,117.728,419.661,171.673,31.768,155.923
C04990=1057.173,117.976,419.641,171.674,31.770,155.924
C04991=1057.178,118.226,419.621,171.676,31.773,155.924
C04992=1057.184,118.475,419.601,171.677,31.776,155.924
C04993=1057.191,118.725,419.581,171.679,31.778,155.925
C04994=1057.197,118.973,419.561,171.680,31.781,155.925
C04995=1057.202,119.222,419.541,171.682,31.784,155.926
C04996=1057.208,119.471,419.521,171.684,31.786,155.926
C04997=1057.214,119.720,419.501,171.686,31.788,155.926
C04998=1057.220,119.970,419.480,171.688,31.791,155.927
C04999=1057.225,120.219,419.461,171.689,31.793,155.927
C05000=1057.231,120.468,419.441,171.691,31.796,155.928
C05001=1057.237,120.717,419.421,171.692,31.799,155.928
C05002=1057.243,120.967,419.400,171.694,31.801,155.928
C05003=1057.249,121.216,419.380,171.695,31.803,155.929
C05004=1057.255,121.464,419.360,171.697,31.806,155.929
C05005=1057.261,121.713,419.340,171.699,31.808,155.930
C05006=1057.267,121.963,419.319,171.701,31.811,155.930
C05007=1057.273,122.212,419.299,171.703,31.814,155.930
C05008=1057.279,122.461,419.279,171.704,31.816,155.931
C05009=1057.285,122.711,419.258,171.706,31.818,155.931
C05010=1057.291,122.959,419.238,171.708,31.821,155.932
C05011=1057.297,123.208,419.218,171.709,31.824,155.932
C05012=1057.303,123.457,419.198,171.711,31.826,155.932
C05013=1057.309,123.707,419.177,171.712,31.828,155.933
C05014=1057.315,123.956,419.157,171.714,31.831,155.933
C05015=1057.321,124.204,419.137,171.716,31.833,155.934
C05016=1057.327,124.454,419.116,171.718,31.836,155.934
C05017=1057.333,124.703,419.096,171.720,31.839,155.934
C05018=1057.339,124.952,419.076,171.721,31.841,155.935
C05019=1057.344,125.202,419.056,171.723,31.843,155.935
C05020=1057.350,125.450,419.036,171.724,31.846,155.936
C05021=1057.356,125.699,419.016,171.726,31.848,155.936
C05022=1057.363,125.985,418.992,171.728,31.851,155.936
C05023=1057.370,126.269,418.969,171.730,31.854,155.937
C05024=1057.378,126.554,418.946,171.732,31.857,155.937
C05025=1057.384,126.839,418.922,171.734,31.860,155.938
C05026=1057.391,127.088,418.901,171.736,31.862,155.938
C05027=1057.396,127.337,418.881,171.738,31.865,155.939
C05028=1057.402,127.586,418.861,171.740,31.867,155.939
C05029=1057.409,127.835,418.840,171.741,31.870,155.939
C05030=1057.414,128.085,418.820,171.742,31.872,155.940
C05031=1057.420,128.333,418.800,171.744,31.875,155.940
C05032=1057.427,128.583,418.780,171.746,31.877,155.941
C05033=1057.432,128.831,418.758,171.748,31.879,155.941
C05034=1057.439,129.081,418.738,171.750,31.882,155.941
C05035=1057.444,129.330,418.717,171.751,31.884,155.942
C05036=1057.451,129.580,418.697,171.753,31.887,155.942
C05037=1057.457,129.828,418.676,171.755,31.889,155.943
C05038=1057.462,130.077,418.656,171.757,31.892,155.943
C05039=1057.469,130.326,418.636,171.758,31.894,155.943
C05040=1057.475,130.575,418.616,171.760,31.897,155.944
C05041=1057.481,130.824,418.594,171.762,31.900,155.944
C05042=1057.487,131.073,418.574,171.763,31.902,155.945
C05043=1057.493,131.323,418.554,171.765,31.904,155.945
C05044=1057.499,131.572,418.533,171.767,31.907,155.945
C05045=1057.506,131.821,418.512,171.769,31.909,155.946
C05046=1057.511,132.070,418.492,171.771,31.912,155.946
C05047=1057.516,132.319,418.471,171.773,31.914,155.947
C05048=1057.523,132.568,418.450,171.774,31.917,155.947
C05049=1057.528,132.817,418.429,171.775,31.919,155.947
C05050=1057.535,133.067,418.409,171.777,31.922,155.948
C05051=1057.540,133.315,418.388,171.779,31.925,155.948
C05052=1057.546,133.564,418.367,171.781,31.927,155.949
C05053=1057.553,133.813,418.346,171.783,31.930,155.949
C05054=1057.558,134.062,418.326,171.784,31.932,155.950
C05055=1057.564,134.312,418.305,171.786,31.935,155.950
C05056=1057.570,134.560,418.284,171.788,31.938,155.950
C05057=1057.576,134.810,418.263,171.790,31.940,155.951
C05058=1057.582,135.058,418.243,171.792,31.942,155.951
C05059=1057.588,135.308,418.222,171.793,31.945,155.952
C05060=1057.594,135.557,418.200,171.795,31.947,155.952
C05061=1057.600,135.805,418.180,171.796,31.950,155.952
C05062=1057.606,136.055,418.159,171.798,31.953,155.953
C05063=1057.611,136.304,418.138,171.800,31.955,155.953
C05064=1057.618,136.553,418.117,171.802,31.958,155.954
C05065=1057.623,136.802,418.097,171.804,31.960,155.954
C05066=1057.629,137.051,418.075,171.806,31.962,155.954
C05067=1057.635,137.300,418.055,171.808,31.965,155.955
C05068=1057.641,137.549,418.033,171.809,31.968,155.955
C05069=1057.647,137.798,418.013,171.811,31.970,155.956
C05070=1057.654,138.047,417.992,171.812,31.973,155.956
C05071=1057.659,138.296,417.971,171.814,31.975,155.957
C05072=1057.665,138.545,417.950,171.816,31.978,155.957
C05073=1057.670,138.794,417.929,171.818,31.981,155.957
C05074=1057.677,139.043,417.908,171.820,31.983,155.958
C05075=1057.683,139.292,417.887,171.822,31.985,155.958
C05076=1057.689,139.542,417.866,171.823,31.988,155.959
C05077=1057.695,139.791,417.844,171.825,31.990,155.959
C05078=1057.701,140.040,417.824,171.827,31.993,155.959
C05079=1057.707,140.289,417.803,171.829,31.996,155.960
C05080=1057.712,140.537,417.781,171.830,31.998,155.960
C05081=1057.718,140.787,417.760,171.832,32.001,155.961
C05082=1057.724,141.036,417.739,171.834,32.004,155.961
C05083=1057.730,141.285,417.717,171.836,32.006,155.961
C05084=1057.735,141.534,417.697,171.837,32.009,155.962
C05085=1057.741,141.783,417.675,171.839,32.011,155.962
C05086=1057.748,142.067,417.651,171.841,32.015,155.963
C05087=1057.756,142.352,417.627,171.844,32.017,155.963
C05088=1057.762,142.638,417.603,171.846,32.020,155.964
C05089=1057.768,142.922,417.579,171.848,32.023,155.964
C05090=1057.775,143.171,417.557,171.849,32.026,155.965
C05091=1057.780,143.420,417.536,171.851,32.028,155.965
C05092=1057.786,143.669,417.515,171.853,32.031,155.966
C05093=1057.792,143.919,417.493,171.855,32.034,155.966
C05094=1057.798,144.167,417.472,171.856,32.036,155.966
C05095=1057.805,144.416,417.451,171.858,32.039,155.967
C05096=1057.810,144.665,417.430,171.860,32.041,155.967
C05097=1057.816,144.914,417.409,171.862,32.044,155.968
C05098=1057.822,145.164,417.387,171.864,32.047,155.968
C05099=1057.828,145.412,417.366,171.866,32.049,155.968
C05100=1057.834,145.661,417.344,171.868,32.052,155.969
C05101=1057.840,145.910,417.323,171.869,32.054,155.969
C05102=1057.845,146.160,417.302,171.871,32.056,155.970
C05103=1057.852,146.409,417.280,171.873,32.059,155.970
C05104=1057.857,146.657,417.259,171.875,32.062,155.970
C05105=1057.863,146.906,417.237,171.876,32.064,155.971
C05106=1057.869,147.156,417.216,171.878,32.067,155.971
C05107=1057.875,147.404,417.195,171.880,32.069,155.972
C05108=1057.881,147.653,417.173,171.882,32.072,155.972
C05109=1057.887,147.903,417.151,171.884,32.075,155.973
C05110=1057.893,148.151,417.130,171.886,32.077,155.973
C05111=1057.899,148.400,417.108,171.888,32.080,155.973
C05112=1057.905,148.650,417.087,171.889,32.082,155.974
C05113=1057.911,148.898,417.065,171.891,32.085,155.974
C05114=1057.917,149.147,417.044,171.893,32.088,155.975
C05115=1057.923,149.396,417.023,171.895,32.090,155.975
C05116=1057.929,149.645,417.001,171.897,32.093,155.976
C05117=1057.935,149.894,416.979,171.899,32.095,155.976
C05118=1057.940,150.143,416.958,171.900,32.098,155.976
C05119=1057.946,150.392,416.936,171.902,32.101,155.977
C05120=1057.952,150.641,416.914,171.904,32.103,155.977
C05121=1057.958,150.891,416.892,171.906,32.106,155.978
C05122=1057.964,151.139,416.871,171.908,32.108,155.978
C05123=1057.970,151.388,416.850,171.910,32.111,155.979
C05124=1057.976,151.637,416.828,171.911,32.114,155.979
C05125=1057.981,151.886,416.806,171.913,32.116,155.979
C05126=1057.987,152.135,416.784,171.915,32.119,155.980
C05127=1057.993,152.385,416.763,171.917,32.122,155.980
C05128=1057.999,152.633,416.742,171.919,32.125,155.981
C05129=1058.005,152.882,416.720,171.921,32.127,155.981
C05130=1058.011,153.131,416.698,171.923,32.130,155.982
C05131=1058.017,153.381,416.675,171.925,32.132,155.982
C05132=1058.022,153.629,416.654,171.927,32.135,155.983
C05133=1058.029,153.878,416.632,171.929,32.138,155.983
C05134=1058.035,154.127,416.611,171.931,32.140,155.983
C05135=1058.040,154.376,416.590,171.932,32.143,155.984
C05136=1058.046,154.625,416.567,171.933,32.145,155.984
C05137=1058.052,154.874,416.545,171.935,32.148,155.985
C05138=1058.058,155.123,416.523,171.937,32.151,155.985
C05139=1058.064,155.372,416.502,171.939,32.153,155.986
C05140=1058.069,155.621,416.480,171.941,32.156,155.986
C05141=1058.076,155.870,416.457,171.943,32.158,155.986
C05142=1058.082,156.119,416.436,171.945,32.161,155.987
C05143=1058.087,156.368,416.414,171.947,32.164,155.987
C05144=1058.093,156.616,416.392,171.949,32.166,155.988
C05145=1058.099,156.866,416.370,171.951,32.169,155.988
C05146=1058.105,157.115,416.348,171.953,32.172,155.989
C05147=1058.111,157.364,416.326,171.954,32.175,155.989
C05148=1058.117,157.612,416.304,171.956,32.177,155.989
C05149=1058.122,157.862,416.282,171.958,32.180,155.990
C05150=1058.130,158.146,416.257,171.960,32.183,155.990
C05151=1058.136,158.431,416.232,171.963,32.186,155.991
C05152=1058.143,158.715,416.207,171.965,32.189,155.991
C05153=1058.149,159.000,416.182,171.967,32.192,155.992
C05154=1058.156,159.248,416.159,171.969,32.195,155.992
C05155=1058.162,159.498,416.138,171.971,32.197,155.993
C05156=1058.167,159.747,416.115,171.973,32.200,155.993
C05157=1058.173,159.995,416.093,171.975,32.203,155.994
C05158=1058.179,160.245,416.071,171.977,32.205,155.994
C05159=1058.185,160.493,416.049,171.978,32.208,155.995
C05160=1058.191,160.742,416.027,171.980,32.210,155.995
C05161=1058.197,160.991,416.004,171.982,32.213,155.995
C05162=1058.203,161.240,415.983,171.984,32.216,155.996
C05163=1058.208,161.489,415.960,171.986,32.219,155.996
C05164=1058.214,161.738,415.938,171.988,32.221,155.997
C05165=1058.220,161.987,415.915,171.990,32.224,155.997
C05166=1058.226,162.236,415.893,171.992,32.227,155.998
C05167=1058.231,162.484,415.871,171.994,32.230,155.998
C05168=1058.236,162.734,415.848,171.996,32.232,155.999
C05169=1058.243,162.983,415.826,171.998,32.235,155.999
C05170=1058.248,163.232,415.804,172.000,32.238,156.000
C05171=1058.254,163.481,415.781,172.002,32.241,156.000
C05172=1058.260,163.729,415.759,172.003,32.243,156.000
C05173=1058.265,163.978,415.737,172.005,32.246,156.001
C05174=1058.271,164.227,415.714,172.007,32.249,156.001
C05175=1058.276,164.477,415.691,172.009,32.252,156.002
C05176=1058.283,164.725,415.669,172.011,32.254,156.002
C05177=1058.288,164.974,415.646,172.013,32.257,156.003
C05178=1058.293,165.223,415.624,172.015,32.260,156.003
C05179=1058.300,165.472,415.602,172.017,32.263,156.004
C05180=1058.306,165.721,415.579,172.019,32.266,156.004
C05181=1058.311,165.970,415.557,172.021,32.268,156.005
C05182=1058.317,166.219,415.534,172.023,32.271,156.005
C05183=1058.323,166.468,415.511,172.025,32.274,156.005
C05184=1058.329,166.717,415.489,172.027,32.277,156.006
C05185=1058.334,166.966,415.466,172.028,32.279,156.006
C05186=1058.339,167.214,415.444,172.030,32.282,156.007
C05187=1058.346,167.463,415.421,172.032,32.285,156.007
C05188=1058.351,167.712,415.399,172.034,32.288,156.008
C05189=1058.357,167.961,415.376,172.036,32.290,156.008
C05190=1058.363,168.210,415.353,172.038,32.293,156.009
C05191=1058.369,168.459,415.331,172.041,32.296,156.009
C05192=1058.375,168.708,415.309,172.043,32.299,156.010
C05193=1058.380,168.957,415.286,172.045,32.301,156.010
C05194=1058.386,169.206,415.263,172.047,32.304,156.011
C05195=1058.392,169.455,415.240,172.049,32.307,156.011
C05196=1058.398,169.703,415.217,172.051,32.310,156.012
C05197=1058.404,169.952,415.195,172.053,32.312,156.012
C05198=1058.409,170.202,415.172,172.054,32.315,156.012
C05199=1058.415,170.451,415.149,172.056,32.318,156.013
C05200=1058.421,170.699,415.127,172.058,32.321,156.013
C05201=1058.427,170.948,415.104,172.060,32.323,156.014
C05202=1058.433,171.196,415.081,172.062,32.327,156.014
C05203=1058.438,171.445,415.059,172.064,32.329,156.015
C05204=1058.444,171.694,415.036,172.066,32.332,156.015
C05205=1058.450,171.943,415.013,172.068,32.334,156.016
C05206=1058.456,172.192,414.991,172.070,32.337,156.016
C05207=1058.462,172.441,414.968,172.073,32.340,156.017
C05208=1058.467,172.690,414.945,172.075,32.343,156.017
C05209=1058.473,172.939,414.922,172.077,32.345,156.017
C05210=1058.479,173.189,414.899,172.079,32.349,156.018
C05211=1058.486,173.437,414.876,172.081,32.351,156.018
C05212=1058.492,173.686,414.854,172.082,32.354,156.019
C05213=1058.497,173.935,414.831,172.084,32.357,156.019
C05214=1058.504,174.218,414.805,172.086,32.359,156.020
C05215=1058.511,174.503,414.779,172.089,32.363,156.020
C05216=1058.517,174.787,414.752,172.091,32.366,156.021
C05217=1058.524,175.071,414.726,172.094,32.369,156.021
C05218=1058.530,175.320,414.703,172.096,32.372,156.022
C05219=1058.536,175.569,414.680,172.098,32.375,156.022
C05220=1058.542,175.818,414.658,172.100,32.378,156.023
C05221=1058.548,176.066,414.635,172.102,32.380,156.023
C05222=1058.554,176.315,414.612,172.104,32.383,156.024
C05223=1058.560,176.564,414.588,172.106,32.386,156.024
C05224=1058.566,176.813,414.565,172.108,32.388,156.025
C05225=1058.572,177.062,414.542,172.111,32.391,156.025
C05226=1058.577,177.311,414.519,172.113,32.394,156.026
C05227=1058.584,177.560,414.497,172.114,32.397,156.026
C05228=1058.590,177.808,414.474,172.116,32.400,156.026
C05229=1058.595,178.057,414.451,172.118,32.402,156.027
C05230=1058.601,178.306,414.428,172.120,32.405,156.027
C05231=1058.608,178.555,414.404,172.122,32.408,156.028
C05232=1058.613,178.804,414.381,172.124,32.410,156.028
C05233=1058.619,179.053,414.358,172.127,32.414,156.029
C05234=1058.625,179.302,414.335,172.129,32.416,156.029
C05235=1058.631,179.550,414.313,172.131,32.419,156.030
C05236=1058.637,179.799,414.289,172.133,32.421,156.030
C05237=1058.644,180.048,414.266,172.135,32.425,156.031
C05238=1058.649,180.297,414.243,172.137,32.427,156.031
C05239=1058.655,180.546,414.220,172.140,32.430,156.032
C05240=1058.661,180.794,414.196,172.142,32.433,156.032
C05241=1058.668,181.044,414.173,172.144,32.436,156.033
C05242=1058.673,181.293,414.150,172.145,32.438,156.033
C05243=1058.679,181.542,414.127,172.147,32.441,156.033
C05244=1058.686,181.790,414.104,172.149,32.444,156.034
C05245=1058.692,182.039,414.081,172.152,32.447,156.034
C05246=1058.698,182.288,414.058,172.154,32.449,156.035
C05247=1058.704,182.537,414.034,172.156,32.452,156.035
C05248=1058.710,182.785,414.011,172.158,32.455,156.036
C05249=1058.715,183.034,413.988,172.160,32.458,156.036
C05250=1058.722,183.283,413.964,172.162,32.460,156.037
C05251=1058.728,183.532,413.941,172.165,32.463,156.037
C05252=1058.734,183.781,413.918,172.167,32.466,156.038
C05253=1058.740,184.030,413.894,172.169,32.469,156.038
C05254=1058.746,184.279,413.871,172.171,32.472,156.039
C05255=1058.752,184.527,413.848,172.173,32.474,156.039
C05256=1058.758,184.776,413.825,172.176,32.478,156.040
C05257=1058.763,185.025,413.800,172.178,32.480,156.040
C05258=1058.769,185.274,413.777,172.180,32.483,156.041
C05259=1058.775,185.523,413.753,172.181,32.486,156.041
C05260=1058.780,185.772,413.730,172.183,32.489,156.042
C05261=1058.786,186.020,413.706,172.185,32.492,156.042
C05262=1058.791,186.269,413.683,172.188,32.495,156.042
C05263=1058.798,186.518,413.659,172.190,32.498,156.043
C05264=1058.804,186.767,413.635,172.192,32.501,156.043
C05265=1058.809,187.016,413.611,172.194,32.504,156.044
C05266=1058.815,187.264,413.588,172.196,32.506,156.044
C05267=1058.821,187.514,413.564,172.198,32.510,156.045
C05268=1058.827,187.762,413.540,172.201,32.513,156.046
C05269=1058.832,188.011,413.516,172.203,32.515,156.046
C05270=1058.838,188.260,413.493,172.205,32.519,156.047
C05271=1058.844,188.508,413.469,172.207,32.521,156.047
C05272=1058.849,188.758,413.445,172.209,32.524,156.048
C05273=1058.855,189.006,413.422,172.212,32.528,156.048
C05274=1058.861,189.255,413.398,172.214,32.530,156.048
C05275=1058.867,189.504,413.374,172.216,32.533,156.049
C05276=1058.872,189.753,413.350,172.218,32.536,156.050
C05277=1058.878,190.001,413.326,172.219,32.539,156.050
C05278=1058.885,190.285,413.299,172.222,32.542,156.051
C05279=1058.892,190.569,413.272,172.225,32.546,156.051
C05280=1058.898,190.853,413.245,172.227,32.549,156.052
C05281=1058.905,191.136,413.218,172.230,32.553,156.052
C05282=1058.911,191.385,413.193,172.232,32.556,156.053
C05283=1058.916,191.634,413.170,172.234,32.558,156.053
C05284=1058.922,191.882,413.146,172.236,32.561,156.054
C05285=1058.928,192.131,413.122,172.239,32.565,156.054
C05286=1058.934,192.380,413.098,172.241,32.567,156.055
C05287=1058.940,192.628,413.074,172.243,32.570,156.055
C05288=1058.946,192.877,413.050,172.245,32.573,156.056
C05289=1058.951,193.126,413.027,172.248,32.576,156.056
C05290=1058.957,193.376,413.002,172.250,32.579,156.057
C05291=1058.963,193.624,412.978,172.252,32.582,156.057
C05292=1058.969,193.872,412.954,172.254,32.585,156.058
C05293=1058.975,194.121,412.930,172.257,32.588,156.058
C05294=1058.981,194.370,412.906,172.259,32.591,156.059
C05295=1058.987,194.619,412.882,172.260,32.594,156.059
C05296=1058.992,194.868,412.857,172.262,32.597,156.060
C05297=1058.998,195.117,412.835,172.265,32.600,156.060
C05298=1059.004,195.366,412.810,172.267,32.603,156.061
C05299=1059.010,195.614,412.786,172.269,32.606,156.061
C05300=1059.016,195.863,412.762,172.271,32.609,156.062
C05301=1059.022,196.112,412.738,172.274,32.612,156.062
C05302=1059.028,196.361,412.713,172.276,32.615,156.063
C05303=1059.034,196.609,412.690,172.278,32.618,156.063
C05304=1059.039,196.858,412.665,172.281,32.621,156.064
C05305=1059.046,197.107,412.641,172.283,32.624,156.064
C05306=1059.051,197.355,412.617,172.285,32.627,156.065
C05307=1059.058,197.604,412.593,172.287,32.630,156.066
C05308=1059.063,197.853,412.569,172.290,32.632,156.066
C05309=1059.070,198.102,412.545,172.292,32.636,156.067
C05310=1059.075,198.351,412.521,172.294,32.639,156.067
C05311=1059.082,198.599,412.496,172.297,32.641,156.067
C05312=1059.087,198.847,412.472,172.299,32.645,156.068
C05313=1059.094,199.096,412.448,172.301,32.648,156.069
C05314=1059.099,199.345,412.423,172.304,32.650,156.069
C05315=1059.106,199.594,412.399,172.306,32.654,156.070
C05316=1059.111,199.843,412.375,172.308,32.657,156.070
C05317=1059.117,200.092,412.350,172.310,32.659,156.071
C05318=1059.124,200.341,412.326,172.312,32.662,156.071
C05319=1059.129,200.589,412.301,172.314,32.666,156.072
C05320=1059.136,200.838,412.277,172.316,32.668,156.072
C05321=1059.141,201.086,412.253,172.319,32.671,156.073
C05322=1059.148,201.335,412.229,172.321,32.675,156.073
C05323=1059.153,201.584,412.205,172.324,32.678,156.074
C05324=1059.159,201.833,412.179,172.326,32.680,156.074
C05325=1059.166,202.082,412.155,172.328,32.684,156.075
C05326=1059.171,202.330,412.131,172.331,32.687,156.075
C05327=1059.177,202.579,412.107,172.333,32.690,156.076
C05328=1059.183,202.827,412.082,172.335,32.693,156.076
C05329=1059.189,203.077,412.057,172.337,32.696,156.077
C05330=1059.195,203.325,412.033,172.340,32.699,156.077
C05331=1059.201,203.574,412.008,172.342,32.702,156.078
C05332=1059.206,203.822,411.984,172.344,32.705,156.078
C05333=1059.212,204.072,411.959,172.347,32.708,156.079
C05334=1059.218,204.320,411.934,172.349,32.711,156.080
C05335=1059.224,204.569,411.910,172.352,32.715,156.080
C05336=1059.230,204.817,411.884,172.354,32.718,156.081
C05337=1059.235,205.066,411.860,172.356,32.721,156.081
C05338=1059.242,205.315,411.836,172.359,32.724,156.082
C05339=1059.248,205.563,411.811,172.361,32.727,156.082
C05340=1059.253,205.812,411.786,172.363,32.730,156.083
C05341=1059.260,206.061,411.761,172.366,32.733,156.083
C05342=1059.285,207.110,411.657,172.551,32.820,156.093
C05343=1059.290,207.342,411.633,172.552,32.823,156.094
C05344=1059.296,207.574,411.610,172.554,32.827,156.095
C05345=1059.302,207.805,411.585,172.556,32.830,156.096
C05346=1059.308,208.038,411.562,172.558,32.834,156.096
C05347=1059.313,208.269,411.537,172.560,32.838,156.097
C05348=1059.319,208.501,411.513,172.562,32.842,156.098
C05349=1059.325,208.732,411.489,172.563,32.846,156.098
C05350=1059.330,208.964,411.466,172.565,32.849,156.099
C05351=1059.336,209.213,411.441,172.567,32.853,156.100
C05352=1059.342,209.461,411.414,172.569,32.857,156.101
C05353=1059.348,209.710,411.389,172.571,32.861,156.101
C05354=1059.355,209.959,411.363,172.573,32.865,156.102
C05355=1059.361,210.207,411.337,172.575,32.869,156.103
C05356=1059.367,210.456,411.311,172.577,32.873,156.103
C05357=1059.373,210.705,411.286,172.579,32.877,156.104
C05358=1059.380,210.953,411.259,172.581,32.881,156.105
C05359=1059.385,211.202,411.234,172.583,32.885,156.106
C05360=1059.392,211.450,411.208,172.585,32.889,156.106
C05361=1059.398,211.699,411.182,172.587,32.893,156.107
C05362=1059.404,211.948,411.156,172.589,32.897,156.108
C05363=1059.410,212.196,411.130,172.591,32.901,156.109
C05364=1059.416,212.445,411.105,172.593,32.904,156.109
C05365=1059.423,212.694,411.078,172.595,32.909,156.110
C05366=1059.429,212.942,411.052,172.597,32.912,156.111
C05367=1059.435,213.191,411.026,172.599,32.917,156.112
C05368=1059.441,213.439,411.001,172.601,32.920,156.112
C05369=1059.447,213.688,410.974,172.603,32.925,156.113
C05370=1059.453,213.936,410.949,172.605,32.928,156.114
C05371=1059.459,214.185,410.922,172.607,32.933,156.115
C05372=1059.465,214.433,410.897,172.609,32.936,156.115
C05373=1059.471,214.681,410.870,172.611,32.940,156.116
C05374=1059.478,214.930,410.843,172.613,32.944,156.117
C05375=1059.484,215.179,410.818,172.615,32.948,156.118
C05376=1059.490,215.428,410.791,172.617,32.952,156.118
C05377=1059.496,215.676,410.766,172.619,32.956,156.119
C05378=1059.502,215.925,410.739,172.621,32.960,156.120
C05379=1059.508,216.173,410.713,172.623,32.964,156.120
C05380=1059.514,216.422,410.687,172.625,32.968,156.121
C05381=1059.521,216.670,410.661,172.627,32.972,156.122
C05382=1059.527,216.919,410.634,172.629,32.976,156.123
C05383=1059.532,217.168,410.609,172.631,32.980,156.123
C05384=1059.539,217.416,410.582,172.633,32.983,156.124
C05385=1059.545,217.665,410.555,172.635,32.987,156.125
C05386=1059.551,217.913,410.530,172.637,32.991,156.126
C05387=1059.557,218.162,410.503,172.639,32.995,156.126
C05388=1059.563,218.410,410.477,172.641,32.999,156.127
C05389=1059.569,218.660,410.451,172.643,33.003,156.128
C05390=1059.576,218.908,410.425,172.645,33.007,156.129
C05391=1059.582,219.156,410.398,172.647,33.011,156.129
C05392=1059.588,219.404,410.372,172.649,33.015,156.130
C05393=1059.594,219.654,410.346,172.651,33.019,156.131
C05394=1059.601,219.902,410.320,172.653,33.022,156.131
C05395=1059.607,220.150,410.293,172.655,33.027,156.132
C05396=1059.612,220.398,410.267,172.657,33.030,156.133
C05397=1059.620,220.647,410.240,172.659,33.034,156.134
C05398=1059.625,220.896,410.214,172.662,33.038,156.134
C05399=1059.631,221.130,410.190,172.664,33.042,156.135
C05400=1059.637,221.364,410.164,172.665,33.045,156.136
C05401=1059.643,221.599,410.140,172.667,33.049,156.136
C05402=1059.648,221.833,410.114,172.669,33.053,156.137
C05403=1059.654,222.067,410.089,172.671,33.056,156.138
C05404=1059.660,222.301,410.065,172.673,33.060,156.139
C05405=1059.665,222.535,410.039,172.675,33.064,156.139
C05406=1059.672,222.770,410.014,172.677,33.067,156.140
C05407=1059.678,223.018,409.987,172.679,33.071,156.141
C05408=1059.683,223.266,409.961,172.681,33.075,156.141
C05409=1059.690,223.516,409.934,172.683,33.079,156.142
C05410=1059.696,223.764,409.907,172.685,33.083,156.143
C05411=1059.702,224.012,409.881,172.687,33.087,156.144
C05412=1059.708,224.261,409.854,172.690,33.091,156.144
C05413=1059.714,224.509,409.827,172.692,33.095,156.145
C05414=1059.720,224.758,409.801,172.694,33.099,156.146
C05415=1059.726,225.007,409.774,172.696,33.103,156.147
C05416=1059.733,225.255,409.748,172.698,33.106,156.147
C05417=1059.739,225.503,409.721,172.700,33.110,156.148
C05418=1059.745,225.752,409.694,172.702,33.114,156.149
C05419=1059.751,226.001,409.667,172.704,33.118,156.149
C05420=1059.757,226.249,409.641,172.706,33.122,156.150
C05421=1059.763,226.498,409.614,172.708,33.126,156.151
C05422=1059.770,226.745,409.587,172.711,33.130,156.152
C05423=1059.776,226.995,409.560,172.713,33.133,156.152
C05424=1059.782,227.243,409.533,172.715,33.138,156.153
C05425=1059.788,227.491,409.507,172.717,33.141,156.154
C05426=1059.794,227.740,409.480,172.719,33.145,156.154
C05427=1059.800,227.989,409.453,172.721,33.149,156.155
C05428=1059.807,228.237,409.426,172.723,33.153,156.156
C05429=1059.813,228.485,409.399,172.725,33.156,156.157
C05430=1059.819,228.734,409.372,172.728,33.160,156.157
C05431=1059.825,228.983,409.346,172.730,33.164,156.158
C05432=1059.832,229.232,409.319,172.732,33.168,156.159
C05433=1059.838,229.479,409.291,172.734,33.172,156.160
C05434=1059.843,229.728,409.265,172.736,33.176,156.160
C05435=1059.850,229.977,409.238,172.738,33.180,156.161
C05436=1059.856,230.225,409.210,172.741,33.183,156.162
C05437=1059.862,230.474,409.183,172.744,33.188,156.163
C05438=1059.868,230.722,409.157,172.746,33.191,156.163
C05439=1059.875,230.970,409.129,172.748,33.195,156.164
C05440=1059.880,231.219,409.102,172.750,33.199,156.165
C05441=1059.887,231.468,409.075,172.752,33.203,156.165
C05442=1059.893,231.716,409.048,172.754,33.207,156.166
C05443=1059.899,231.964,409.021,172.757,33.211,156.167
C05444=1059.905,232.212,408.993,172.759,33.214,156.168
C05445=1059.911,232.461,408.967,172.761,33.218,156.168
C05446=1059.918,232.710,408.940,172.763,33.222,156.169
C05447=1059.924,232.958,408.912,172.765,33.226,156.170
C05448=1059.929,233.207,408.885,172.767,33.230,156.170
C05449=1059.935,233.455,408.857,172.770,33.234,156.171
C05450=1059.942,233.704,408.830,172.772,33.238,156.172
C05451=1059.948,233.951,408.803,172.774,33.241,156.173
C05452=1059.954,234.200,408.776,172.776,33.246,156.173
C05453=1059.960,234.449,408.748,172.778,33.249,156.174
C05454=1059.966,234.698,408.721,172.780,33.253,156.175
C05455=1059.972,234.927,408.696,172.782,33.256,156.176
C05456=1059.977,235.158,408.670,172.784,33.260,156.176
C05457=1059.983,235.389,408.645,172.786,33.264,156.177
C05458=1059.989,235.618,408.620,172.789,33.267,156.178
C05459=1059.994,235.849,408.594,172.791,33.271,156.178
C05460=1060.000,236.079,408.568,172.793,33.275,156.179
C05461=1060.006,236.309,408.544,172.795,33.278,156.180
C05462=1060.012,236.539,408.517,172.797,33.281,156.180
